SPLINE
SPL {X  -115.209, Y  +259.476, Z    +0.000, E1   +49.595, E3 +267374.990}
SPL {X  -147.344, Y  +302.806, Z    +0.000, E1   +40.158, E3 +267464.452}
SPL {X  -160.798, Y  +338.700, Z    +0.000, E1   +25.294, E3 +267463.934}
SPL {X  -163.893, Y  +354.439, Z    +0.000, E1   +16.805, E3 +267458.408}
SPL {X  -165.158, Y  +365.746, Z    +0.000, E1   +10.198, E3 +267456.351}
SPL {X  -165.639, Y  +376.620, Z    +0.000, E1    +3.186, E3 +267456.151}
SPL {X  -165.650, Y  +380.533, Z    +0.000, E1    +0.120, E3 +267455.179}
SPL {X  -165.650, Y  +383.454, Z    +0.000, E1    -2.667, E3 +267454.586}
SPL {X  -165.650, Y  +388.792, Z    +0.000, E1    -9.482, E3 +267453.680}
SPL {X  -165.650, Y  +393.970, Z    +0.000, E1   -17.146, E3 +267452.837}
SPL {X  -165.650, Y  +401.614, Z    +0.000, E1   -27.619, E3 +267453.492}
SPL {X  -165.650, Y  +418.105, Z    +0.000, E1   -49.413, E3 +267448.900}
SPL {X  -165.650, Y  +465.736, Z    +0.000, E1   -65.678, E3 +267462.642}
SPL {X  -165.650, Y  +519.483, Z    +0.000, E1   -68.357, E3 +267488.827}
SPL {X  -165.650, Y  +548.869, Z    +0.000, E1   -62.199, E3 +267544.519}
ENDSPLINE

SPLINE
SPL {X  -165.650, Y  +534.780, Z    +0.000, E1   -57.803, E3 +267558.169}
ENDSPLINE

SPLINE
SPL {X  -165.650, Y  +545.905, Z    +0.000, E1   -57.853, E3 +267572.108}
SPL {X  -165.650, Y  +553.630, Z    +0.000, E1   -57.616, E3 +267583.558}
SPL {X  -165.650, Y  +563.473, Z    +0.000, E1   -57.690, E3 +267595.922}
SPL {X  -165.650, Y  +573.011, Z    +0.000, E1   -57.610, E3 +267608.713}
SPL {X  -165.650, Y  +581.530, Z    +0.000, E1   -57.678, E3 +267619.311}
SPL {X  -165.650, Y  +589.475, Z    +0.000, E1   -57.572, E3 +267630.298}
SPL {X  -165.650, Y  +599.695, Z    +0.000, E1   -57.964, E3 +267640.914}
SPL {X  -165.650, Y  +606.915, Z    +0.000, E1   -57.651, E3 +267652.271}
SPL {X  -165.650, Y  +614.927, Z    +0.000, E1   -57.517, E3 +267663.541}
SPL {X  -165.650, Y  +624.337, Z    +0.000, E1   -57.671, E3 +267674.767}
SPL {X  -165.650, Y  +634.236, Z    +0.000, E1   -57.671, E3 +267687.617}
SPL {X  -165.650, Y  +644.287, Z    +0.000, E1   -57.872, E3 +267699.183}
SPL {X  -165.650, Y  +650.480, Z    +0.000, E1   -57.669, E3 +267708.488}
SPL {X  -165.650, Y  +657.986, Z    +0.000, E1   -57.646, E3 +267718.380}
SPL {X  -165.650, Y  +667.585, Z    +0.000, E1   -57.803, E3 +267729.776}
SPL {X  -165.650, Y  +673.199, Z    +0.000, E1   -57.412, E3 +267739.520}
SPL {X  -165.558, Y  +681.013, Z    +0.000, E1   -57.768, E3 +267747.359}
SPL {X  -165.167, Y  +688.139, Z    +0.000, E1   -57.463, E3 +267758.657}
SPL {X  -164.323, Y  +696.426, Z    +0.000, E1   -57.565, E3 +267768.644}
SPL {X  -163.313, Y  +703.224, Z    +0.000, E1   -57.403, E3 +267778.538}
SPL {X  -161.906, Y  +710.520, Z    +0.000, E1   -57.149, E3 +267789.489}
SPL {X  -160.577, Y  +716.182, Z    +0.000, E1   -56.676, E3 +267799.750}
SPL {X  -158.520, Y  +723.576, Z    +0.000, E1   -56.758, E3 +267808.795}
SPL {X  -156.858, Y  +728.749, Z    +0.000, E1   -56.333, E3 +267817.937}
SPL {X  -155.155, Y  +733.525, Z    +0.000, E1   -55.869, E3 +267826.714}
SPL {X  -153.442, Y  +737.914, Z    +0.000, E1   -55.562, E3 +267834.118}
SPL {X  -150.574, Y  +744.547, Z    +0.000, E1   -55.310, E3 +267844.101}
SPL {X  -147.713, Y  +750.471, Z    +0.000, E1   -54.514, E3 +267855.764}
SPL {X  -139.786, Y  +764.381, Z    +0.000, E1   -57.209, E3 +267859.952}
SPL {X  -110.324, Y  +799.066, Z    +0.000, E1   -54.396, E3 +267928.526}
SPL {X  -100.308, Y  +807.326, Z    +0.000, E1   -52.880, E3 +267973.093}
ENDSPLINE

SPLINE
SPL {X  -108.196, Y  +800.934, Z    +0.000, E1   -52.068, E3 +268065.420}
SPL {X  -144.673, Y  +756.182, Z    +0.000, E1   -41.752, E3 +268083.499}
SPL {X  -158.838, Y  +722.515, Z    +0.000, E1   -28.697, E3 +268082.983}
SPL {X  -163.562, Y  +701.720, Z    +0.000, E1   -18.114, E3 +268080.196}
SPL {X  -165.078, Y  +689.251, Z    +0.000, E1   -10.876, E3 +268081.748}
SPL {X  -165.596, Y  +679.730, Z    +0.000, E1    -4.777, E3 +268079.267}
SPL {X  -165.650, Y  +674.376, Z    +0.000, E1    -0.866, E3 +268079.183}
SPL {X  -165.650, Y  +672.384, Z    +0.000, E1    +0.908, E3 +268078.064}
SPL {X  -165.650, Y  +669.093, Z    +0.000, E1    +4.549, E3 +268077.915}
SPL {X  -165.650, Y  +663.273, Z    +0.000, E1   +12.448, E3 +268077.152}
SPL {X  -165.650, Y  +654.885, Z    +0.000, E1   +25.204, E3 +268075.704}
SPL {X  -165.650, Y  +641.882, Z    +0.000, E1   +46.566, E3 +268068.575}
SPL {X  -165.650, Y  +630.946, Z    +0.000, E1   +55.779, E3 +268069.250}
SPL {X  -165.650, Y  +595.858, Z    +0.000, E1   +64.262, E3 +268084.131}
SPL {X  -165.650, Y  +589.368, Z    +0.000, E1   +58.232, E3 +268104.872}
SPL {X  -165.650, Y  +491.251, Z    +0.000, E1   +65.373, E3 +268161.299}
ENDSPLINE

SPLINE
SPL {X  -165.650, Y  +516.236, Z    +0.000, E1   +58.457, E3 +268181.979}
ENDSPLINE

SPLINE
SPL {X  -165.650, Y  +506.715, Z    +0.000, E1   +58.090, E3 +268196.432}
SPL {X  -165.650, Y  +496.085, Z    +0.000, E1   +57.984, E3 +268210.680}
SPL {X  -165.650, Y  +485.167, Z    +0.000, E1   +58.003, E3 +268224.512}
ENDSPLINE

SPLINE
SPL {X  -165.650, Y  +509.193, Z    +0.000, E1   +50.604, E3 +268235.478}
ENDSPLINE

SPLINE
SPL {X  -165.650, Y  +503.302, Z    +0.000, E1   +50.402, E3 +268246.575}
SPL {X  -165.650, Y  +495.166, Z    +0.000, E1   +51.070, E3 +268256.152}
SPL {X  -165.650, Y  +485.807, Z    +0.000, E1   +51.973, E3 +268265.885}
SPL {X  -165.650, Y  +478.030, Z    +0.000, E1   +52.389, E3 +268275.691}
SPL {X  -165.650, Y  +467.527, Z    +0.000, E1   +53.334, E3 +268286.186}
SPL {X  -165.650, Y  +457.379, Z    +0.000, E1   +53.935, E3 +268297.729}
SPL {X  -165.650, Y  +444.120, Z    +0.000, E1   +54.815, E3 +268311.775}
SPL {X  -165.650, Y  +431.771, Z    +0.000, E1   +55.549, E3 +268324.604}
SPL {X  -165.650, Y  +420.799, Z    +0.000, E1   +56.452, E3 +268333.990}
SPL {X  -165.650, Y  +409.731, Z    +0.000, E1   +57.273, E3 +268343.479}
SPL {X  -165.650, Y  +399.687, Z    +0.000, E1   +57.433, E3 +268355.663}
SPL {X  -165.650, Y  +388.492, Z    +0.000, E1   +57.709, E3 +268368.376}
SPL {X  -165.650, Y  +379.894, Z    +0.000, E1   +57.709, E3 +268379.480}
SPL {X  -165.538, Y  +372.423, Z    +0.000, E1   +57.528, E3 +268390.353}
SPL {X  -164.865, Y  +362.388, Z    +0.000, E1   +57.628, E3 +268402.739}
SPL {X  -163.867, Y  +354.258, Z    +0.000, E1   +57.359, E3 +268414.956}
SPL {X  -162.678, Y  +347.264, Z    +0.000, E1   +57.150, E3 +268425.298}
SPL {X  -161.618, Y  +342.173, Z    +0.000, E1   +56.783, E3 +268434.183}
SPL {X  -159.878, Y  +335.155, Z    +0.000, E1   +56.685, E3 +268443.987}
SPL {X  -158.009, Y  +328.771, Z    +0.000, E1   +56.325, E3 +268454.346}
SPL {X  -156.065, Y  +322.971, Z    +0.000, E1   +56.177, E3 +268462.690}
SPL {X  -154.487, Y  +318.719, Z    +0.000, E1   +55.733, E3 +268470.699}
SPL {X  -151.902, Y  +312.426, Z    +0.000, E1   +55.494, E3 +268480.174}
SPL {X  -149.742, Y  +307.668, Z    +0.000, E1   +54.896, E3 +268489.386}
SPL {X  -146.487, Y  +301.160, Z    +0.000, E1   +54.808, E3 +268498.249}
SPL {X  -133.590, Y  +280.553, Z    +0.000, E1   +59.642, E3 +268499.206}
SPL {X  -112.638, Y  +257.040, Z    +0.000, E1   +51.417, E3 +268602.589}
ENDSPLINE

SPLINE
SPL {X  -115.209, Y  +259.476, Z    +0.000, E1   +49.595, E3 +268635.859}
SPL {X  -147.344, Y  +302.806, Z    +0.000, E1   +40.158, E3 +268725.322}
SPL {X  -160.798, Y  +338.700, Z    +0.000, E1   +25.294, E3 +268724.804}
SPL {X  -163.893, Y  +354.439, Z    +0.000, E1   +16.805, E3 +268719.278}
SPL {X  -165.158, Y  +365.746, Z    +0.000, E1   +10.198, E3 +268717.220}
SPL {X  -165.580, Y  +373.688, Z    +0.000, E1    +5.094, E3 +268716.957}
SPL {X  -165.650, Y  +379.719, Z    +0.000, E1    +0.894, E3 +268716.387}
SPL {X  -165.650, Y  +383.454, Z    +0.000, E1    -2.667, E3 +268715.455}
SPL {X  -165.650, Y  +387.779, Z    +0.000, E1    -8.159, E3 +268715.129}
SPL {X  -165.650, Y  +392.511, Z    +0.000, E1   -14.940, E3 +268713.620}
SPL {X  -165.650, Y  +401.614, Z    +0.000, E1   -27.619, E3 +268714.361}
SPL {X  -165.650, Y  +417.340, Z    +0.000, E1   -48.811, E3 +268709.663}
SPL {X  -165.650, Y  +462.495, Z    +0.000, E1   -65.156, E3 +268722.495}
SPL {X  -165.650, Y  +519.483, Z    +0.000, E1   -68.357, E3 +268749.696}
SPL {X  -165.650, Y  +548.869, Z    +0.000, E1   -62.199, E3 +268805.389}
ENDSPLINE

SPLINE
SPL {X  -165.650, Y  +534.780, Z    +0.000, E1   -57.803, E3 +268819.038}
ENDSPLINE

SPLINE
SPL {X  -165.650, Y  +545.905, Z    +0.000, E1   -57.853, E3 +268832.978}
SPL {X  -165.650, Y  +553.630, Z    +0.000, E1   -57.616, E3 +268844.427}
SPL {X  -165.650, Y  +563.473, Z    +0.000, E1   -57.690, E3 +268856.791}
SPL {X  -165.650, Y  +573.011, Z    +0.000, E1   -57.610, E3 +268869.583}
SPL {X  -165.650, Y  +581.530, Z    +0.000, E1   -57.678, E3 +268880.181}
SPL {X  -165.650, Y  +589.475, Z    +0.000, E1   -57.572, E3 +268891.168}
SPL {X  -165.650, Y  +599.695, Z    +0.000, E1   -57.964, E3 +268901.784}
SPL {X  -165.650, Y  +606.915, Z    +0.000, E1   -57.651, E3 +268913.140}
SPL {X  -165.650, Y  +614.927, Z    +0.000, E1   -57.517, E3 +268924.410}
SPL {X  -165.650, Y  +624.337, Z    +0.000, E1   -57.671, E3 +268935.636}
SPL {X  -165.650, Y  +634.236, Z    +0.000, E1   -57.671, E3 +268948.486}
SPL {X  -165.650, Y  +647.519, Z    +0.000, E1   -57.817, E3 +268964.814}
SPL {X  -165.650, Y  +657.986, Z    +0.000, E1   -57.646, E3 +268979.249}
SPL {X  -165.650, Y  +667.585, Z    +0.000, E1   -57.803, E3 +268990.645}
SPL {X  -165.634, Y  +677.794, Z    +0.000, E1   -57.650, E3 +269004.947}
SPL {X  -165.167, Y  +688.139, Z    +0.000, E1   -57.463, E3 +269019.527}
SPL {X  -164.009, Y  +698.761, Z    +0.000, E1   -57.613, E3 +269032.300}
SPL {X  -162.382, Y  +708.242, Z    +0.000, E1   -57.205, E3 +269047.226}
SPL {X  -160.577, Y  +716.182, Z    +0.000, E1   -56.676, E3 +269060.619}
SPL {X  -158.520, Y  +723.576, Z    +0.000, E1   -56.758, E3 +269069.664}
SPL {X  -156.858, Y  +728.749, Z    +0.000, E1   -56.333, E3 +269078.807}
SPL {X  -155.155, Y  +733.525, Z    +0.000, E1   -55.869, E3 +269087.583}
SPL {X  -153.442, Y  +737.914, Z    +0.000, E1   -55.562, E3 +269094.988}
SPL {X  -150.574, Y  +744.547, Z    +0.000, E1   -55.310, E3 +269104.971}
SPL {X  -147.713, Y  +750.471, Z    +0.000, E1   -54.514, E3 +269116.633}
SPL {X  -139.786, Y  +764.381, Z    +0.000, E1   -57.209, E3 +269120.821}
SPL {X  -110.324, Y  +799.066, Z    +0.000, E1   -54.396, E3 +269189.396}
SPL {X  -100.308, Y  +807.326, Z    +0.000, E1   -52.880, E3 +269233.963}
ENDSPLINE

SPLINE
SPL {X  -108.196, Y  +800.934, Z    +0.000, E1   -52.068, E3 +269326.289}
SPL {X  -144.673, Y  +756.182, Z    +0.000, E1   -41.752, E3 +269344.368}
SPL {X  -158.838, Y  +722.515, Z    +0.000, E1   -28.697, E3 +269343.852}
SPL {X  -163.562, Y  +701.720, Z    +0.000, E1   -18.114, E3 +269341.066}
SPL {X  -165.380, Y  +684.954, Z    +0.000, E1    -8.247, E3 +269341.248}
SPL {X  -165.650, Y  +675.104, Z    +0.000, E1    -1.512, E3 +269340.043}
SPL {X  -165.650, Y  +672.384, Z    +0.000, E1    +0.908, E3 +269338.933}
SPL {X  -165.650, Y  +669.968, Z    +0.000, E1    +3.584, E3 +269338.749}
SPL {X  -165.650, Y  +666.667, Z    +0.000, E1    +7.761, E3 +269338.428}
SPL {X  -165.650, Y  +662.028, Z    +0.000, E1   +14.359, E3 +269338.058}
SPL {X  -165.650, Y  +654.885, Z    +0.000, E1   +25.204, E3 +269336.574}
SPL {X  -165.650, Y  +641.882, Z    +0.000, E1   +46.566, E3 +269329.445}
SPL {X  -165.650, Y  +630.946, Z    +0.000, E1   +55.779, E3 +269330.119}
SPL {X  -165.650, Y  +590.135, Z    +0.000, E1   +59.110, E3 +269362.739}
SPL {X  -165.650, Y  +491.251, Z    +0.000, E1   +65.373, E3 +269422.168}
ENDSPLINE

SPLINE
SPL {X  -165.650, Y  +516.236, Z    +0.000, E1   +58.457, E3 +269442.849}
ENDSPLINE

SPLINE
SPL {X  -165.650, Y  +506.715, Z    +0.000, E1   +58.090, E3 +269457.302}
SPL {X  -165.650, Y  +496.085, Z    +0.000, E1   +57.984, E3 +269471.549}
SPL {X  -165.650, Y  +485.167, Z    +0.000, E1   +58.003, E3 +269485.381}
ENDSPLINE

SPLINE
SPL {X  -165.650, Y  +505.180, Z    +0.000, E1   +52.333, E3 +269492.133}
SPL {X  -165.650, Y  +506.534, Z    +0.000, E1   +50.148, E3 +269503.593}
ENDSPLINE

SPLINE
SPL {X  -165.650, Y  +495.166, Z    +0.000, E1   +51.070, E3 +269517.021}
SPL {X  -165.650, Y  +485.807, Z    +0.000, E1   +51.973, E3 +269526.754}
SPL {X  -165.650, Y  +475.672, Z    +0.000, E1   +52.573, E3 +269539.208}
SPL {X  -165.650, Y  +459.814, Z    +0.000, E1   +53.888, E3 +269555.397}
SPL {X  -165.650, Y  +448.876, Z    +0.000, E1   +54.452, E3 +269567.892}
SPL {X  -165.650, Y  +440.843, Z    +0.000, E1   +55.023, E3 +269575.956}
SPL {X  -165.650, Y  +431.771, Z    +0.000, E1   +55.549, E3 +269585.474}
SPL {X  -165.650, Y  +420.799, Z    +0.000, E1   +56.452, E3 +269594.860}
SPL {X  -165.650, Y  +409.731, Z    +0.000, E1   +57.273, E3 +269604.348}
SPL {X  -165.650, Y  +399.687, Z    +0.000, E1   +57.433, E3 +269616.533}
SPL {X  -165.650, Y  +388.492, Z    +0.000, E1   +57.709, E3 +269629.246}
SPL {X  -165.650, Y  +379.894, Z    +0.000, E1   +57.709, E3 +269640.350}
SPL {X  -165.538, Y  +372.423, Z    +0.000, E1   +57.528, E3 +269651.222}
SPL {X  -164.865, Y  +362.388, Z    +0.000, E1   +57.628, E3 +269663.609}
SPL {X  -163.867, Y  +354.258, Z    +0.000, E1   +57.359, E3 +269675.826}
SPL {X  -162.678, Y  +347.264, Z    +0.000, E1   +57.150, E3 +269686.167}
SPL {X  -161.618, Y  +342.173, Z    +0.000, E1   +56.783, E3 +269695.053}
SPL {X  -159.878, Y  +335.155, Z    +0.000, E1   +56.685, E3 +269704.856}
SPL {X  -158.009, Y  +328.771, Z    +0.000, E1   +56.325, E3 +269715.216}
SPL {X  -156.065, Y  +322.971, Z    +0.000, E1   +56.177, E3 +269723.560}
SPL {X  -153.731, Y  +316.803, Z    +0.000, E1   +55.737, E3 +269734.136}
SPL {X  -150.320, Y  +308.902, Z    +0.000, E1   +55.085, E3 +269747.832}
SPL {X  -146.487, Y  +301.160, Z    +0.000, E1   +54.808, E3 +269759.118}
SPL {X  -133.590, Y  +280.553, Z    +0.000, E1   +59.642, E3 +269760.075}
SPL {X  -112.638, Y  +257.040, Z    +0.000, E1   +51.417, E3 +269863.459}
ENDSPLINE

SPLINE
SPL {X  -115.209, Y  +259.476, Z    +0.000, E1   +49.595, E3 +269896.729}
SPL {X  -147.344, Y  +302.806, Z    +0.000, E1   +40.158, E3 +269986.191}
SPL {X  -160.798, Y  +338.700, Z    +0.000, E1   +25.294, E3 +269985.673}
SPL {X  -163.893, Y  +354.439, Z    +0.000, E1   +16.805, E3 +269980.147}
SPL {X  -165.158, Y  +365.746, Z    +0.000, E1   +10.198, E3 +269978.090}
SPL {X  -165.639, Y  +376.620, Z    +0.000, E1    +3.186, E3 +269977.890}
SPL {X  -165.650, Y  +380.533, Z    +0.000, E1    +0.120, E3 +269976.918}
SPL {X  -165.650, Y  +382.353, Z    +0.000, E1    -1.616, E3 +269976.499}
SPL {X  -165.650, Y  +386.363, Z    +0.000, E1    -6.162, E3 +269976.049}
SPL {X  -165.650, Y  +392.511, Z    +0.000, E1   -14.940, E3 +269974.489}
SPL {X  -165.650, Y  +401.614, Z    +0.000, E1   -27.619, E3 +269975.231}
SPL {X  -165.650, Y  +418.105, Z    +0.000, E1   -49.413, E3 +269970.639}
SPL {X  -165.650, Y  +465.736, Z    +0.000, E1   -65.678, E3 +269984.381}
SPL {X  -165.650, Y  +519.483, Z    +0.000, E1   -68.357, E3 +270010.566}
SPL {X  -165.650, Y  +548.869, Z    +0.000, E1   -62.199, E3 +270066.259}
ENDSPLINE

SPLINE
SPL {X  -165.650, Y  +534.780, Z    +0.000, E1   -57.803, E3 +270079.908}
ENDSPLINE

SPLINE
SPL {X  -165.650, Y  +545.905, Z    +0.000, E1   -57.853, E3 +270093.847}
SPL {X  -165.650, Y  +555.746, Z    +0.000, E1   -57.571, E3 +270108.485}
SPL {X  -165.650, Y  +566.557, Z    +0.000, E1   -57.834, E3 +270120.613}
SPL {X  -165.650, Y  +573.011, Z    +0.000, E1   -57.610, E3 +270130.452}
SPL {X  -165.650, Y  +581.530, Z    +0.000, E1   -57.678, E3 +270141.050}
SPL {X  -165.650, Y  +589.475, Z    +0.000, E1   -57.572, E3 +270152.037}
SPL {X  -165.650, Y  +599.695, Z    +0.000, E1   -57.964, E3 +270162.653}
SPL {X  -165.650, Y  +606.915, Z    +0.000, E1   -57.651, E3 +270174.010}
SPL {X  -165.650, Y  +614.927, Z    +0.000, E1   -57.517, E3 +270185.280}
SPL {X  -165.650, Y  +624.337, Z    +0.000, E1   -57.671, E3 +270196.506}
SPL {X  -165.650, Y  +634.236, Z    +0.000, E1   -57.671, E3 +270209.356}
SPL {X  -165.650, Y  +644.287, Z    +0.000, E1   -57.872, E3 +270220.922}
SPL {X  -165.650, Y  +650.480, Z    +0.000, E1   -57.669, E3 +270230.227}
SPL {X  -165.650, Y  +657.986, Z    +0.000, E1   -57.646, E3 +270240.119}
SPL {X  -165.650, Y  +667.585, Z    +0.000, E1   -57.803, E3 +270251.515}
SPL {X  -165.650, Y  +673.199, Z    +0.000, E1   -57.412, E3 +270261.259}
SPL {X  -165.558, Y  +681.013, Z    +0.000, E1   -57.768, E3 +270269.098}
SPL {X  -165.167, Y  +688.139, Z    +0.000, E1   -57.463, E3 +270280.396}
SPL {X  -164.009, Y  +698.761, Z    +0.000, E1   -57.613, E3 +270293.169}
SPL {X  -162.382, Y  +708.242, Z    +0.000, E1   -57.205, E3 +270308.095}
SPL {X  -160.577, Y  +716.182, Z    +0.000, E1   -56.676, E3 +270321.489}
SPL {X  -158.520, Y  +723.576, Z    +0.000, E1   -56.758, E3 +270330.534}
SPL {X  -156.858, Y  +728.749, Z    +0.000, E1   -56.333, E3 +270339.676}
SPL {X  -155.155, Y  +733.525, Z    +0.000, E1   -55.869, E3 +270348.453}
SPL {X  -152.530, Y  +740.111, Z    +0.000, E1   -55.545, E3 +270358.929}
SPL {X  -149.838, Y  +746.130, Z    +0.000, E1   -55.135, E3 +270368.649}
SPL {X  -147.713, Y  +750.471, Z    +0.000, E1   -54.514, E3 +270377.503}
SPL {X  -139.786, Y  +764.381, Z    +0.000, E1   -57.209, E3 +270381.691}
SPL {X  -110.324, Y  +799.066, Z    +0.000, E1   -54.396, E3 +270450.265}
SPL {X  -100.308, Y  +807.326, Z    +0.000, E1   -52.880, E3 +270494.832}
ENDSPLINE

SPLINE
SPL {X  -108.196, Y  +800.934, Z    +0.000, E1   -52.068, E3 +270587.159}
SPL {X  -147.753, Y  +750.393, Z    +0.000, E1   -39.863, E3 +270605.381}
SPL {X  -161.414, Y  +712.720, Z    +0.000, E1   -24.024, E3 +270604.723}
SPL {X  -164.278, Y  +696.774, Z    +0.000, E1   -15.225, E3 +270599.335}
SPL {X  -165.380, Y  +684.954, Z    +0.000, E1    -8.247, E3 +270602.118}
SPL {X  -165.650, Y  +675.104, Z    +0.000, E1    -1.512, E3 +270600.913}
SPL {X  -165.650, Y  +672.384, Z    +0.000, E1    +0.908, E3 +270599.803}
SPL {X  -165.650, Y  +669.093, Z    +0.000, E1    +4.549, E3 +270599.654}
SPL {X  -165.650, Y  +663.273, Z    +0.000, E1   +12.448, E3 +270598.891}
SPL {X  -165.650, Y  +657.199, Z    +0.000, E1   +21.720, E3 +270598.161}
SPL {X  -165.650, Y  +652.963, Z    +0.000, E1   +28.395, E3 +270596.846}
SPL {X  -165.650, Y  +641.882, Z    +0.000, E1   +46.566, E3 +270590.314}
SPL {X  -165.650, Y  +630.946, Z    +0.000, E1   +55.779, E3 +270590.989}
SPL {X  -165.650, Y  +590.135, Z    +0.000, E1   +59.110, E3 +270623.609}
SPL {X  -165.650, Y  +491.251, Z    +0.000, E1   +65.373, E3 +270683.038}
ENDSPLINE

SPLINE
SPL {X  -165.650, Y  +516.236, Z    +0.000, E1   +58.457, E3 +270703.718}
ENDSPLINE

SPLINE
SPL {X  -165.650, Y  +506.715, Z    +0.000, E1   +58.090, E3 +270718.171}
SPL {X  -165.650, Y  +496.085, Z    +0.000, E1   +57.984, E3 +270732.419}
SPL {X  -165.650, Y  +485.167, Z    +0.000, E1   +58.003, E3 +270746.251}
ENDSPLINE

SPLINE
SPL {X  -165.650, Y  +509.193, Z    +0.000, E1   +50.604, E3 +270757.218}
ENDSPLINE

SPLINE
SPL {X  -165.650, Y  +503.302, Z    +0.000, E1   +50.402, E3 +270768.314}
SPL {X  -165.650, Y  +495.166, Z    +0.000, E1   +51.070, E3 +270777.891}
SPL {X  -165.650, Y  +485.807, Z    +0.000, E1   +51.973, E3 +270787.624}
SPL {X  -165.650, Y  +478.030, Z    +0.000, E1   +52.389, E3 +270797.431}
SPL {X  -165.650, Y  +467.527, Z    +0.000, E1   +53.334, E3 +270807.925}
SPL {X  -165.650, Y  +457.379, Z    +0.000, E1   +53.935, E3 +270819.468}
SPL {X  -165.650, Y  +444.120, Z    +0.000, E1   +54.815, E3 +270833.514}
SPL {X  -165.650, Y  +431.771, Z    +0.000, E1   +55.549, E3 +270846.344}
SPL {X  -165.650, Y  +420.799, Z    +0.000, E1   +56.452, E3 +270855.729}
SPL {X  -165.650, Y  +409.731, Z    +0.000, E1   +57.273, E3 +270865.218}
SPL {X  -165.650, Y  +399.687, Z    +0.000, E1   +57.433, E3 +270877.402}
SPL {X  -165.650, Y  +388.492, Z    +0.000, E1   +57.709, E3 +270890.115}
SPL {X  -165.650, Y  +379.894, Z    +0.000, E1   +57.709, E3 +270901.219}
SPL {X  -165.538, Y  +372.423, Z    +0.000, E1   +57.528, E3 +270912.092}
SPL {X  -164.865, Y  +362.388, Z    +0.000, E1   +57.628, E3 +270924.478}
SPL {X  -163.867, Y  +354.258, Z    +0.000, E1   +57.359, E3 +270936.695}
SPL {X  -162.678, Y  +347.264, Z    +0.000, E1   +57.150, E3 +270947.037}
SPL {X  -161.618, Y  +342.173, Z    +0.000, E1   +56.783, E3 +270955.922}
SPL {X  -159.878, Y  +335.155, Z    +0.000, E1   +56.685, E3 +270965.726}
SPL {X  -158.009, Y  +328.771, Z    +0.000, E1   +56.325, E3 +270976.086}
SPL {X  -156.065, Y  +322.971, Z    +0.000, E1   +56.177, E3 +270984.429}
SPL {X  -154.487, Y  +318.719, Z    +0.000, E1   +55.733, E3 +270992.438}
SPL {X  -151.902, Y  +312.426, Z    +0.000, E1   +55.494, E3 +271001.913}
SPL {X  -149.742, Y  +307.668, Z    +0.000, E1   +54.896, E3 +271011.125}
SPL {X  -146.487, Y  +301.160, Z    +0.000, E1   +54.808, E3 +271019.988}
SPL {X  -133.590, Y  +280.553, Z    +0.000, E1   +59.642, E3 +271020.945}
SPL {X  -112.638, Y  +257.040, Z    +0.000, E1   +51.417, E3 +271124.328}
ENDSPLINE

SPLINE
SPL {X  -115.209, Y  +259.476, Z    +0.000, E1   +49.595, E3 +271157.599}
SPL {X  -147.344, Y  +302.806, Z    +0.000, E1   +40.158, E3 +271247.061}
SPL {X  -160.798, Y  +338.700, Z    +0.000, E1   +25.294, E3 +271246.543}
SPL {X  -163.893, Y  +354.439, Z    +0.000, E1   +16.805, E3 +271241.017}
SPL {X  -165.158, Y  +365.746, Z    +0.000, E1   +10.198, E3 +271238.959}
SPL {X  -165.580, Y  +373.688, Z    +0.000, E1    +5.094, E3 +271238.696}
SPL {X  -165.650, Y  +378.140, Z    +0.000, E1    +1.996, E3 +271238.783}
SPL {X  -165.650, Y  +381.477, Z    +0.000, E1    -0.622, E3 +271237.570}
SPL {X  -165.650, Y  +384.861, Z    +0.000, E1    -4.465, E3 +271236.973}
SPL {X  -165.650, Y  +388.792, Z    +0.000, E1    -9.482, E3 +271236.289}
SPL {X  -165.650, Y  +396.421, Z    +0.000, E1   -20.352, E3 +271236.086}
SPL {X  -165.650, Y  +404.249, Z    +0.000, E1   -31.650, E3 +271235.465}
SPL {X  -165.650, Y  +417.340, Z    +0.000, E1   -48.811, E3 +271231.402}
SPL {X  -165.650, Y  +462.495, Z    +0.000, E1   -65.156, E3 +271244.234}
SPL {X  -165.650, Y  +519.483, Z    +0.000, E1   -68.357, E3 +271271.436}
SPL {X  -165.650, Y  +548.869, Z    +0.000, E1   -62.199, E3 +271327.128}
ENDSPLINE

SPLINE
SPL {X  -165.650, Y  +530.735, Z    +0.000, E1   -57.778, E3 +271335.552}
ENDSPLINE

SPLINE
SPL {X  -165.650, Y  +536.777, Z    +0.000, E1   -57.774, E3 +271343.429}
SPL {X  -165.650, Y  +545.905, Z    +0.000, E1   -57.853, E3 +271354.717}
SPL {X  -165.650, Y  +553.630, Z    +0.000, E1   -57.616, E3 +271366.166}
SPL {X  -165.650, Y  +563.473, Z    +0.000, E1   -57.690, E3 +271378.531}
SPL {X  -165.650, Y  +573.011, Z    +0.000, E1   -57.610, E3 +271391.322}
SPL {X  -165.650, Y  +581.530, Z    +0.000, E1   -57.678, E3 +271401.920}
SPL {X  -165.650, Y  +589.475, Z    +0.000, E1   -57.572, E3 +271412.907}
SPL {X  -165.650, Y  +599.695, Z    +0.000, E1   -57.964, E3 +271423.523}
SPL {X  -165.650, Y  +606.915, Z    +0.000, E1   -57.651, E3 +271434.880}
SPL {X  -165.650, Y  +614.927, Z    +0.000, E1   -57.517, E3 +271446.149}
SPL {X  -165.650, Y  +624.337, Z    +0.000, E1   -57.671, E3 +271457.375}
SPL {X  -165.650, Y  +634.236, Z    +0.000, E1   -57.671, E3 +271470.226}
SPL {X  -165.650, Y  +647.519, Z    +0.000, E1   -57.817, E3 +271486.553}
SPL {X  -165.650, Y  +657.986, Z    +0.000, E1   -57.646, E3 +271500.988}
SPL {X  -165.650, Y  +667.585, Z    +0.000, E1   -57.803, E3 +271512.384}
SPL {X  -165.634, Y  +677.794, Z    +0.000, E1   -57.650, E3 +271526.686}
SPL {X  -165.167, Y  +688.139, Z    +0.000, E1   -57.463, E3 +271541.266}
SPL {X  -164.009, Y  +698.761, Z    +0.000, E1   -57.613, E3 +271554.039}
SPL {X  -162.382, Y  +708.242, Z    +0.000, E1   -57.205, E3 +271568.965}
SPL {X  -160.577, Y  +716.182, Z    +0.000, E1   -56.676, E3 +271582.359}
SPL {X  -158.520, Y  +723.576, Z    +0.000, E1   -56.758, E3 +271591.403}
SPL {X  -156.858, Y  +728.749, Z    +0.000, E1   -56.333, E3 +271600.546}
SPL {X  -155.155, Y  +733.525, Z    +0.000, E1   -55.869, E3 +271609.323}
SPL {X  -153.442, Y  +737.914, Z    +0.000, E1   -55.562, E3 +271616.727}
SPL {X  -150.574, Y  +744.547, Z    +0.000, E1   -55.310, E3 +271626.710}
SPL {X  -148.396, Y  +749.110, Z    +0.000, E1   -54.616, E3 +271636.003}
SPL {X  -146.339, Y  +753.120, Z    +0.000, E1   -54.477, E3 +271641.889}
SPL {X  -137.656, Y  +767.645, Z    +0.000, E1   -58.229, E3 +271641.599}
SPL {X  -110.324, Y  +799.066, Z    +0.000, E1   -54.396, E3 +271711.135}
SPL {X  -100.308, Y  +807.326, Z    +0.000, E1   -52.880, E3 +271755.702}
ENDSPLINE

SPLINE
SPL {X  -108.196, Y  +800.934, Z    +0.000, E1   -52.068, E3 +271848.028}
SPL {X  -147.753, Y  +750.393, Z    +0.000, E1   -39.863, E3 +271866.251}
SPL {X  -161.414, Y  +712.720, Z    +0.000, E1   -24.024, E3 +271865.593}
SPL {X  -164.278, Y  +696.774, Z    +0.000, E1   -15.225, E3 +271860.205}
SPL {X  -165.380, Y  +684.954, Z    +0.000, E1    -8.247, E3 +271862.988}
SPL {X  -165.650, Y  +675.104, Z    +0.000, E1    -1.512, E3 +271861.782}
SPL {X  -165.650, Y  +672.384, Z    +0.000, E1    +0.908, E3 +271860.672}
SPL {X  -165.650, Y  +669.968, Z    +0.000, E1    +3.584, E3 +271860.488}
SPL {X  -165.650, Y  +666.667, Z    +0.000, E1    +7.761, E3 +271860.167}
SPL {X  -165.650, Y  +662.028, Z    +0.000, E1   +14.359, E3 +271859.797}
SPL {X  -165.650, Y  +654.885, Z    +0.000, E1   +25.204, E3 +271858.313}
SPL {X  -165.650, Y  +641.882, Z    +0.000, E1   +46.566, E3 +271851.184}
SPL {X  -165.650, Y  +630.946, Z    +0.000, E1   +55.779, E3 +271851.859}
SPL {X  -165.650, Y  +590.135, Z    +0.000, E1   +59.110, E3 +271884.478}
SPL {X  -165.650, Y  +491.251, Z    +0.000, E1   +65.373, E3 +271943.907}
ENDSPLINE

SPLINE
SPL {X  -165.650, Y  +516.236, Z    +0.000, E1   +58.457, E3 +271964.588}
ENDSPLINE

SPLINE
SPL {X  -165.650, Y  +506.715, Z    +0.000, E1   +58.090, E3 +271979.041}
SPL {X  -165.650, Y  +499.697, Z    +0.000, E1   +57.857, E3 +271989.384}
SPL {X  -165.650, Y  +493.307, Z    +0.000, E1   +58.045, E3 +271996.342}
SPL {X  -165.650, Y  +485.167, Z    +0.000, E1   +58.003, E3 +272007.120}
ENDSPLINE

SPLINE
SPL {X  -165.650, Y  +505.180, Z    +0.000, E1   +52.333, E3 +272013.872}
SPL {X  -165.650, Y  +506.534, Z    +0.000, E1   +50.148, E3 +272025.332}
ENDSPLINE

SPLINE
SPL {X  -165.650, Y  +495.166, Z    +0.000, E1   +51.070, E3 +272038.760}
SPL {X  -165.650, Y  +485.807, Z    +0.000, E1   +51.973, E3 +272048.493}
SPL {X  -165.650, Y  +478.030, Z    +0.000, E1   +52.389, E3 +272058.300}
SPL {X  -165.650, Y  +467.527, Z    +0.000, E1   +53.334, E3 +272068.794}
SPL {X  -165.650, Y  +457.379, Z    +0.000, E1   +53.935, E3 +272080.338}
SPL {X  -165.650, Y  +444.120, Z    +0.000, E1   +54.815, E3 +272094.383}
SPL {X  -165.650, Y  +431.771, Z    +0.000, E1   +55.549, E3 +272107.213}
SPL {X  -165.650, Y  +420.799, Z    +0.000, E1   +56.452, E3 +272116.599}
SPL {X  -165.650, Y  +409.731, Z    +0.000, E1   +57.273, E3 +272126.087}
SPL {X  -165.650, Y  +399.687, Z    +0.000, E1   +57.433, E3 +272138.272}
SPL {X  -165.650, Y  +388.492, Z    +0.000, E1   +57.709, E3 +272150.985}
SPL {X  -165.650, Y  +379.894, Z    +0.000, E1   +57.709, E3 +272162.089}
SPL {X  -165.538, Y  +372.423, Z    +0.000, E1   +57.528, E3 +272172.961}
SPL {X  -164.865, Y  +362.388, Z    +0.000, E1   +57.628, E3 +272185.348}
SPL {X  -163.867, Y  +354.258, Z    +0.000, E1   +57.359, E3 +272197.565}
SPL {X  -162.678, Y  +347.264, Z    +0.000, E1   +57.150, E3 +272207.906}
SPL {X  -161.618, Y  +342.173, Z    +0.000, E1   +56.783, E3 +272216.792}
SPL {X  -159.878, Y  +335.155, Z    +0.000, E1   +56.685, E3 +272226.595}
SPL {X  -158.009, Y  +328.771, Z    +0.000, E1   +56.325, E3 +272236.955}
SPL {X  -156.065, Y  +322.971, Z    +0.000, E1   +56.177, E3 +272245.299}
SPL {X  -154.487, Y  +318.719, Z    +0.000, E1   +55.733, E3 +272253.308}
SPL {X  -151.902, Y  +312.426, Z    +0.000, E1   +55.494, E3 +272262.783}
SPL {X  -148.935, Y  +305.985, Z    +0.000, E1   +54.737, E3 +272275.159}
SPL {X  -144.791, Y  +298.030, Z    +0.000, E1   +55.214, E3 +272282.892}
SPL {X  -133.590, Y  +280.553, Z    +0.000, E1   +59.642, E3 +272281.814}
SPL {X  -112.638, Y  +257.040, Z    +0.000, E1   +51.417, E3 +272385.198}
ENDSPLINE

SPLINE
SPL {X  -115.209, Y  +259.476, Z    +0.000, E1   +49.595, E3 +272418.468}
SPL {X  -147.344, Y  +302.806, Z    +0.000, E1   +40.158, E3 +272507.930}
SPL {X  -160.798, Y  +338.700, Z    +0.000, E1   +25.294, E3 +272507.412}
SPL {X  -163.893, Y  +354.439, Z    +0.000, E1   +16.805, E3 +272501.886}
SPL {X  -165.158, Y  +365.746, Z    +0.000, E1   +10.198, E3 +272499.829}
SPL {X  -165.639, Y  +376.620, Z    +0.000, E1    +3.186, E3 +272499.629}
SPL {X  -165.650, Y  +380.533, Z    +0.000, E1    +0.120, E3 +272498.657}
SPL {X  -165.650, Y  +383.454, Z    +0.000, E1    -2.667, E3 +272498.064}
SPL {X  -165.650, Y  +388.792, Z    +0.000, E1    -9.482, E3 +272497.158}
SPL {X  -165.650, Y  +396.421, Z    +0.000, E1   -20.352, E3 +272496.956}
SPL {X  -165.650, Y  +404.249, Z    +0.000, E1   -31.650, E3 +272496.335}
SPL {X  -165.650, Y  +418.105, Z    +0.000, E1   -49.413, E3 +272492.378}
SPL {X  -165.650, Y  +465.736, Z    +0.000, E1   -65.678, E3 +272506.120}
SPL {X  -165.650, Y  +519.483, Z    +0.000, E1   -68.357, E3 +272532.305}
SPL {X  -165.650, Y  +548.869, Z    +0.000, E1   -62.199, E3 +272587.998}
ENDSPLINE

SPLINE
SPL {X  -165.650, Y  +530.735, Z    +0.000, E1   -57.778, E3 +272596.421}
ENDSPLINE

SPLINE
SPL {X  -165.650, Y  +536.777, Z    +0.000, E1   -57.774, E3 +272604.298}
SPL {X  -165.650, Y  +545.905, Z    +0.000, E1   -57.853, E3 +272615.586}
SPL {X  -165.650, Y  +553.630, Z    +0.000, E1   -57.616, E3 +272627.036}
SPL {X  -165.650, Y  +563.473, Z    +0.000, E1   -57.690, E3 +272639.400}
SPL {X  -165.650, Y  +573.011, Z    +0.000, E1   -57.610, E3 +272652.191}
SPL {X  -165.650, Y  +581.530, Z    +0.000, E1   -57.678, E3 +272662.789}
SPL {X  -165.650, Y  +589.475, Z    +0.000, E1   -57.572, E3 +272673.776}
SPL {X  -165.650, Y  +599.695, Z    +0.000, E1   -57.964, E3 +272684.392}
SPL {X  -165.650, Y  +606.915, Z    +0.000, E1   -57.651, E3 +272695.749}
SPL {X  -165.650, Y  +614.927, Z    +0.000, E1   -57.517, E3 +272707.019}
SPL {X  -165.650, Y  +624.337, Z    +0.000, E1   -57.671, E3 +272718.245}
SPL {X  -165.650, Y  +634.236, Z    +0.000, E1   -57.671, E3 +272731.095}
SPL {X  -165.650, Y  +647.519, Z    +0.000, E1   -57.817, E3 +272747.422}
SPL {X  -165.650, Y  +657.986, Z    +0.000, E1   -57.646, E3 +272761.858}
SPL {X  -165.650, Y  +667.585, Z    +0.000, E1   -57.803, E3 +272773.254}
SPL {X  -165.634, Y  +677.794, Z    +0.000, E1   -57.650, E3 +272787.556}
SPL {X  -165.167, Y  +688.139, Z    +0.000, E1   -57.463, E3 +272802.135}
SPL {X  -164.323, Y  +696.426, Z    +0.000, E1   -57.565, E3 +272812.122}
SPL {X  -163.313, Y  +703.224, Z    +0.000, E1   -57.403, E3 +272822.016}
SPL {X  -161.906, Y  +710.520, Z    +0.000, E1   -57.149, E3 +272832.967}
SPL {X  -160.577, Y  +716.182, Z    +0.000, E1   -56.676, E3 +272843.228}
SPL {X  -158.520, Y  +723.576, Z    +0.000, E1   -56.758, E3 +272852.273}
SPL {X  -156.858, Y  +728.749, Z    +0.000, E1   -56.333, E3 +272861.416}
SPL {X  -155.155, Y  +733.525, Z    +0.000, E1   -55.869, E3 +272870.192}
SPL {X  -153.442, Y  +737.914, Z    +0.000, E1   -55.562, E3 +272877.597}
SPL {X  -150.574, Y  +744.547, Z    +0.000, E1   -55.310, E3 +272887.579}
SPL {X  -147.713, Y  +750.471, Z    +0.000, E1   -54.514, E3 +272899.242}
SPL {X  -139.786, Y  +764.381, Z    +0.000, E1   -57.209, E3 +272903.430}
SPL {X  -110.324, Y  +799.066, Z    +0.000, E1   -54.396, E3 +272972.004}
SPL {X  -100.308, Y  +807.326, Z    +0.000, E1   -52.880, E3 +273016.571}
ENDSPLINE

SPLINE
SPL {X  -108.196, Y  +800.934, Z    +0.000, E1   -52.068, E3 +273108.898}
SPL {X  -144.673, Y  +756.182, Z    +0.000, E1   -41.752, E3 +273126.977}
SPL {X  -158.838, Y  +722.515, Z    +0.000, E1   -28.697, E3 +273126.461}
SPL {X  -163.562, Y  +701.720, Z    +0.000, E1   -18.114, E3 +273123.675}
SPL {X  -165.078, Y  +689.251, Z    +0.000, E1   -10.876, E3 +273125.226}
SPL {X  -165.596, Y  +679.730, Z    +0.000, E1    -4.777, E3 +273122.745}
SPL {X  -165.650, Y  +674.376, Z    +0.000, E1    -0.866, E3 +273122.661}
SPL {X  -165.650, Y  +672.384, Z    +0.000, E1    +0.908, E3 +273121.542}
SPL {X  -165.650, Y  +669.093, Z    +0.000, E1    +4.549, E3 +273121.393}
SPL {X  -165.650, Y  +663.273, Z    +0.000, E1   +12.448, E3 +273120.631}
SPL {X  -165.650, Y  +654.885, Z    +0.000, E1   +25.204, E3 +273119.182}
SPL {X  -165.650, Y  +641.882, Z    +0.000, E1   +46.566, E3 +273112.053}
SPL {X  -165.650, Y  +630.946, Z    +0.000, E1   +55.779, E3 +273112.728}
SPL {X  -165.650, Y  +595.858, Z    +0.000, E1   +64.262, E3 +273127.609}
SPL {X  -165.650, Y  +589.368, Z    +0.000, E1   +58.232, E3 +273148.350}
SPL {X  -165.650, Y  +491.251, Z    +0.000, E1   +65.373, E3 +273204.777}
ENDSPLINE

SPLINE
SPL {X  -165.650, Y  +516.236, Z    +0.000, E1   +58.457, E3 +273225.458}
ENDSPLINE

SPLINE
SPL {X  -165.650, Y  +506.715, Z    +0.000, E1   +58.090, E3 +273239.911}
SPL {X  -165.650, Y  +496.085, Z    +0.000, E1   +57.984, E3 +273254.158}
SPL {X  -165.650, Y  +485.167, Z    +0.000, E1   +58.003, E3 +273267.990}
ENDSPLINE

SPLINE
SPL {X  -165.650, Y  +509.193, Z    +0.000, E1   +50.604, E3 +273278.957}
ENDSPLINE

SPLINE
SPL {X  -165.650, Y  +503.302, Z    +0.000, E1   +50.402, E3 +273290.053}
SPL {X  -165.650, Y  +495.166, Z    +0.000, E1   +51.070, E3 +273299.630}
SPL {X  -165.650, Y  +485.807, Z    +0.000, E1   +51.973, E3 +273309.363}
SPL {X  -165.650, Y  +478.030, Z    +0.000, E1   +52.389, E3 +273319.170}
SPL {X  -165.650, Y  +467.527, Z    +0.000, E1   +53.334, E3 +273329.664}
SPL {X  -165.650, Y  +457.379, Z    +0.000, E1   +53.935, E3 +273341.207}
SPL {X  -165.650, Y  +444.120, Z    +0.000, E1   +54.815, E3 +273355.253}
SPL {X  -165.650, Y  +431.771, Z    +0.000, E1   +55.549, E3 +273368.083}
SPL {X  -165.650, Y  +420.799, Z    +0.000, E1   +56.452, E3 +273377.469}
SPL {X  -165.650, Y  +406.746, Z    +0.000, E1   +57.489, E3 +273389.513}
ENDSPLINE

SPLINE
SPL {X  -165.650, Y  +413.842, Z    +0.000, E1   +53.687, E3 +273403.647}
ENDSPLINE

SPLINE
SPL {X  -165.650, Y  +405.379, Z    +0.000, E1   +53.922, E3 +273414.760}
SPL {X  -165.650, Y  +400.791, Z    +0.000, E1   +53.827, E3 +273422.173}
SPL {X  -165.650, Y  +391.401, Z    +0.000, E1   +53.934, E3 +273435.773}
SPL {X  -165.650, Y  +378.987, Z    +0.000, E1   +53.974, E3 +273453.969}
SPL {X  -165.408, Y  +369.556, Z    +0.000, E1   +53.942, E3 +273468.061}
SPL {X  -164.927, Y  +363.041, Z    +0.000, E1   +53.687, E3 +273479.356}
SPL {X  -163.980, Y  +355.035, Z    +0.000, E1   +53.657, E3 +273491.553}
SPL {X  -162.665, Y  +347.197, Z    +0.000, E1   +53.396, E3 +273504.816}
SPL {X  -161.218, Y  +340.437, Z    +0.000, E1   +53.207, E3 +273515.915}
SPL {X  -159.523, Y  +333.864, Z    +0.000, E1   +52.908, E3 +273527.537}
SPL {X  -157.624, Y  +327.563, Z    +0.000, E1   +52.705, E3 +273537.946}
SPL {X  -156.289, Y  +323.602, Z    +0.000, E1   +52.159, E3 +273546.835}
SPL {X  -153.877, Y  +317.168, Z    +0.000, E1   +51.945, E3 +273557.696}
SPL {X  -151.035, Y  +310.467, Z    +0.000, E1   +51.312, E3 +273570.942}
SPL {X  -139.567, Y  +289.276, Z    +0.000, E1   +56.334, E3 +273575.030}
SPL {X  -117.053, Y  +261.289, Z    +0.000, E1   +49.815, E3 +273688.564}
ENDSPLINE

SPLINE
SPL {X  -148.836, Y  +305.783, Z    +0.000, E1   +38.029, E3 +273780.041}
SPL {X  -161.816, Y  +343.065, Z    +0.000, E1   +22.147, E3 +273770.691}
SPL {X  -164.614, Y  +360.007, Z    +0.000, E1   +13.213, E3 +273766.478}
SPL {X  -165.520, Y  +371.933, Z    +0.000, E1    +6.276, E3 +273769.232}
SPL {X  -165.650, Y  +380.164, Z    +0.000, E1    +0.707, E3 +273767.701}
SPL {X  -165.650, Y  +384.850, Z    +0.000, E1    -3.598, E3 +273766.809}
SPL {X  -165.650, Y  +391.255, Z    +0.000, E1   -11.346, E3 +273765.150}
SPL {X  -165.650, Y  +398.038, Z    +0.000, E1   -20.113, E3 +273766.117}
SPL {X  -165.650, Y  +403.005, Z    +0.000, E1   -26.762, E3 +273765.299}
SPL {X  -165.650, Y  +415.469, Z    +0.000, E1   -43.461, E3 +273760.122}
SPL {X  -165.650, Y  +460.095, Z    +0.000, E1   -60.221, E3 +273778.383}
SPL {X  -165.650, Y  +535.749, Z    +0.000, E1   -60.559, E3 +273849.227}
ENDSPLINE

SPLINE
SPL {X  -165.650, Y  +516.750, Z    +0.000, E1   -54.244, E3 +273865.077}
ENDSPLINE

SPLINE
SPL {X  -165.650, Y  +524.345, Z    +0.000, E1   -54.115, E3 +273876.974}
SPL {X  -165.650, Y  +531.171, Z    +0.000, E1   -54.075, E3 +273887.413}
SPL {X  -165.650, Y  +538.771, Z    +0.000, E1   -53.840, E3 +273900.153}
SPL {X  -165.650, Y  +548.103, Z    +0.000, E1   -53.944, E3 +273913.500}
SPL {X  -165.650, Y  +558.071, Z    +0.000, E1   -53.870, E3 +273928.840}
SPL {X  -165.650, Y  +568.053, Z    +0.000, E1   -54.124, E3 +273942.018}
SPL {X  -165.650, Y  +577.021, Z    +0.000, E1   -53.813, E3 +273957.517}
SPL {X  -165.650, Y  +587.996, Z    +0.000, E1   -53.969, E3 +273972.754}
SPL {X  -165.650, Y  +595.185, Z    +0.000, E1   -53.962, E3 +273983.464}
SPL {X  -165.650, Y  +602.138, Z    +0.000, E1   -53.941, E3 +273993.958}
SPL {X  -165.650, Y  +610.307, Z    +0.000, E1   -53.995, E3 +274005.806}
SPL {X  -165.650, Y  +617.878, Z    +0.000, E1   -53.838, E3 +274018.062}
SPL {X  -165.650, Y  +626.374, Z    +0.000, E1   -54.092, E3 +274029.078}
SPL {X  -165.650, Y  +632.964, Z    +0.000, E1   -53.887, E3 +274040.205}
SPL {X  -165.650, Y  +640.262, Z    +0.000, E1   -53.965, E3 +274050.520}
SPL {X  -165.650, Y  +647.911, Z    +0.000, E1   -53.930, E3 +274062.274}
SPL {X  -165.650, Y  +656.836, Z    +0.000, E1   -54.184, E3 +274073.806}
SPL {X  -165.650, Y  +659.513, Z    +0.000, E1   -53.578, E3 +274081.536}
SPL {X  -165.650, Y  +667.820, Z    +0.000, E1   -53.975, E3 +274091.601}
SPL {X  -165.623, Y  +678.503, Z    +0.000, E1   -53.932, E3 +274107.953}
SPL {X  -165.171, Y  +688.090, Z    +0.000, E1   -54.025, E3 +274121.400}
SPL {X  -164.558, Y  +694.489, Z    +0.000, E1   -53.745, E3 +274132.750}
SPL {X  -163.580, Y  +701.606, Z    +0.000, E1   -53.591, E3 +274144.183}
SPL {X  -162.702, Y  +706.614, Z    +0.000, E1   -53.230, E3 +274153.849}
SPL {X  -160.941, Y  +714.715, Z    +0.000, E1   -53.321, E3 +274165.469}
SPL {X  -159.638, Y  +719.723, Z    +0.000, E1   -52.685, E3 +274176.471}
SPL {X  -157.868, Y  +725.674, Z    +0.000, E1   -52.862, E3 +274184.328}
SPL {X  -156.314, Y  +730.327, Z    +0.000, E1   -52.199, E3 +274195.010}
SPL {X  -153.975, Y  +736.588, Z    +0.000, E1   -51.877, E3 +274206.040}
SPL {X  -151.949, Y  +741.465, Z    +0.000, E1   -51.645, E3 +274214.445}
SPL {X  -149.075, Y  +747.727, Z    +0.000, E1   -52.134, E3 +274221.160}
SPL {X  -137.775, Y  +767.467, Z    +0.000, E1   -56.912, E3 +274223.823}
SPL {X  -128.847, Y  +779.607, Z    +0.000, E1   -49.118, E3 +274298.840}
SPL {X   -94.133, Y  +811.804, Z    +0.000, E1   -53.019, E3 +274353.474}
ENDSPLINE

SPLINE
SPL {X  -123.886, Y  +785.464, Z    +0.000, E1   -49.465, E3 +274438.500}
SPL {X  -152.385, Y  +740.452, Z    +0.000, E1   -34.821, E3 +274419.477}
SPL {X  -162.077, Y  +709.719, Z    +0.000, E1   -21.590, E3 +274421.324}
SPL {X  -164.499, Y  +694.994, Z    +0.000, E1   -13.860, E3 +274422.108}
SPL {X  -165.513, Y  +682.236, Z    +0.000, E1    -6.385, E3 +274420.444}
SPL {X  -165.650, Y  +675.776, Z    +0.000, E1    -2.014, E3 +274419.752}
SPL {X  -165.650, Y  +672.041, Z    +0.000, E1    +0.844, E3 +274418.700}
SPL {X  -165.650, Y  +667.328, Z    +0.000, E1    +5.806, E3 +274418.076}
SPL {X  -165.650, Y  +661.774, Z    +0.000, E1   +13.006, E3 +274416.400}
SPL {X  -165.650, Y  +654.085, Z    +0.000, E1   +23.232, E3 +274416.260}
SPL {X  -165.650, Y  +639.700, Z    +0.000, E1   +43.326, E3 +274410.387}
SPL {X  -165.650, Y  +605.320, Z    +0.000, E1   +76.562, E3 +274389.796}
SPL {X  -165.650, Y  +597.745, Z    +0.000, E1   +59.636, E3 +274427.798}
SPL {X  -165.650, Y  +596.360, Z    +0.000, E1   +54.978, E3 +274441.406}
SPL {X  -165.650, Y  +524.050, Z    +0.000, E1   +59.300, E3 +274503.312}
ENDSPLINE

SPLINE
SPL {X  -165.650, Y  +539.856, Z    +0.000, E1   +53.398, E3 +274518.959}
ENDSPLINE

SPLINE
SPL {X  -165.650, Y  +532.042, Z    +0.000, E1   +53.611, E3 +274529.430}
SPL {X  -165.650, Y  +523.239, Z    +0.000, E1   +53.520, E3 +274543.526}
SPL {X  -165.650, Y  +515.134, Z    +0.000, E1   +53.252, E3 +274557.255}
SPL {X  -165.650, Y  +505.685, Z    +0.000, E1   +53.701, E3 +274568.863}
SPL {X  -165.650, Y  +498.275, Z    +0.000, E1   +53.357, E3 +274582.170}
SPL {X  -165.650, Y  +491.031, Z    +0.000, E1   +53.348, E3 +274593.190}
SPL {X  -165.650, Y  +479.077, Z    +0.000, E1   +55.039, E3 +274600.313}
SPL {X  -165.650, Y  +450.615, Z    +0.000, E1   +59.721, E3 +274606.819}
SPL {X  -165.650, Y  +449.326, Z    +0.000, E1   +58.606, E3 +274615.868}
SPL {X  -165.650, Y  +442.154, Z    +0.000, E1   +58.369, E3 +274626.492}
SPL {X  -165.650, Y  +437.405, Z    +0.000, E1   +57.663, E3 +274637.102}
SPL {X  -165.650, Y  +432.227, Z    +0.000, E1   +57.103, E3 +274647.590}
SPL {X  -165.650, Y  +428.683, Z    +0.000, E1   +56.222, E3 +274657.944}
SPL {X  -165.650, Y  +424.202, Z    +0.000, E1   +55.382, E3 +274669.633}
SPL {X  -165.650, Y  +418.469, Z    +0.000, E1   +54.594, E3 +274682.741}
SPL {X  -165.650, Y  +413.857, Z    +0.000, E1   +53.683, E3 +274695.312}
SPL {X  -165.650, Y  +405.379, Z    +0.000, E1   +53.922, E3 +274706.426}
SPL {X  -165.650, Y  +400.791, Z    +0.000, E1   +53.827, E3 +274713.840}
SPL {X  -165.650, Y  +393.046, Z    +0.000, E1   +53.951, E3 +274724.732}
SPL {X  -165.650, Y  +383.306, Z    +0.000, E1   +53.987, E3 +274739.010}
SPL {X  -165.640, Y  +376.676, Z    +0.000, E1   +53.760, E3 +274750.176}
SPL {X  -165.408, Y  +369.556, Z    +0.000, E1   +53.942, E3 +274759.727}
SPL {X  -164.927, Y  +363.041, Z    +0.000, E1   +53.687, E3 +274771.023}
SPL {X  -164.096, Y  +355.862, Z    +0.000, E1   +53.838, E3 +274780.753}
SPL {X  -163.142, Y  +349.785, Z    +0.000, E1   +53.493, E3 +274791.969}
SPL {X  -161.604, Y  +342.113, Z    +0.000, E1   +53.155, E3 +274805.463}
SPL {X  -160.424, Y  +337.221, Z    +0.000, E1   +52.694, E3 +274815.303}
SPL {X  -158.192, Y  +329.354, Z    +0.000, E1   +52.890, E3 +274826.135}
SPL {X  -156.289, Y  +323.602, Z    +0.000, E1   +52.159, E3 +274838.502}
SPL {X  -154.898, Y  +319.792, Z    +0.000, E1   +51.850, E3 +274845.837}
SPL {X  -152.682, Y  +314.249, Z    +0.000, E1   +51.841, E3 +274854.234}
SPL {X  -150.607, Y  +309.525, Z    +0.000, E1   +51.147, E3 +274864.719}
SPL {X  -139.567, Y  +289.276, Z    +0.000, E1   +56.334, E3 +274866.697}
SPL {X  -117.053, Y  +261.289, Z    +0.000, E1   +49.815, E3 +274980.230}
ENDSPLINE

SPLINE
SPL {X  -148.836, Y  +305.783, Z    +0.000, E1   +38.029, E3 +275071.708}
SPL {X  -161.816, Y  +343.065, Z    +0.000, E1   +22.147, E3 +275062.358}
SPL {X  -164.614, Y  +360.007, Z    +0.000, E1   +13.213, E3 +275058.144}
SPL {X  -165.520, Y  +371.933, Z    +0.000, E1    +6.276, E3 +275060.899}
SPL {X  -165.650, Y  +378.704, Z    +0.000, E1    +1.700, E3 +275059.768}
SPL {X  -165.650, Y  +382.197, Z    +0.000, E1    -1.038, E3 +275058.841}
SPL {X  -165.650, Y  +386.782, Z    +0.000, E1    -5.783, E3 +275058.319}
SPL {X  -165.650, Y  +392.406, Z    +0.000, E1   -13.042, E3 +275056.216}
SPL {X  -165.650, Y  +398.038, Z    +0.000, E1   -20.113, E3 +275057.784}
SPL {X  -165.650, Y  +403.005, Z    +0.000, E1   -26.762, E3 +275056.966}
SPL {X  -165.650, Y  +415.469, Z    +0.000, E1   -43.461, E3 +275051.789}
SPL {X  -165.650, Y  +460.095, Z    +0.000, E1   -60.221, E3 +275070.050}
SPL {X  -165.650, Y  +537.366, Z    +0.000, E1   -61.810, E3 +275134.626}
ENDSPLINE

SPLINE
SPL {X  -165.650, Y  +520.647, Z    +0.000, E1   -55.836, E3 +275152.318}
ENDSPLINE

SPLINE
SPL {X  -165.650, Y  +521.328, Z    +0.000, E1   -53.870, E3 +275165.735}
SPL {X  -165.650, Y  +531.171, Z    +0.000, E1   -54.075, E3 +275179.079}
SPL {X  -165.650, Y  +538.771, Z    +0.000, E1   -53.840, E3 +275191.820}
SPL {X  -165.650, Y  +548.103, Z    +0.000, E1   -53.944, E3 +275205.166}
SPL {X  -165.650, Y  +558.071, Z    +0.000, E1   -53.870, E3 +275220.507}
SPL {X  -165.650, Y  +568.053, Z    +0.000, E1   -54.124, E3 +275233.685}
SPL {X  -165.650, Y  +574.396, Z    +0.000, E1   -53.807, E3 +275245.076}
SPL {X  -165.650, Y  +579.991, Z    +0.000, E1   -53.716, E3 +275253.986}
SPL {X  -165.650, Y  +587.996, Z    +0.000, E1   -53.969, E3 +275264.421}
SPL {X  -165.650, Y  +595.185, Z    +0.000, E1   -53.962, E3 +275275.130}
SPL {X  -165.650, Y  +602.138, Z    +0.000, E1   -53.941, E3 +275285.625}
SPL {X  -165.650, Y  +610.307, Z    +0.000, E1   -53.995, E3 +275297.472}
SPL {X  -165.650, Y  +617.878, Z    +0.000, E1   -53.838, E3 +275309.729}
SPL {X  -165.650, Y  +626.374, Z    +0.000, E1   -54.092, E3 +275320.744}
SPL {X  -165.650, Y  +632.964, Z    +0.000, E1   -53.887, E3 +275331.872}
SPL {X  -165.650, Y  +640.262, Z    +0.000, E1   -53.965, E3 +275342.187}
SPL {X  -165.650, Y  +647.911, Z    +0.000, E1   -53.930, E3 +275353.941}
SPL {X  -165.650, Y  +656.836, Z    +0.000, E1   -54.184, E3 +275365.473}
SPL {X  -165.650, Y  +659.513, Z    +0.000, E1   -53.578, E3 +275373.203}
SPL {X  -165.650, Y  +667.820, Z    +0.000, E1   -53.975, E3 +275383.268}
SPL {X  -165.623, Y  +678.503, Z    +0.000, E1   -53.932, E3 +275399.619}
SPL {X  -165.027, Y  +689.850, Z    +0.000, E1   -53.862, E3 +275416.883}
SPL {X  -163.840, Y  +699.919, Z    +0.000, E1   -53.732, E3 +275432.665}
SPL {X  -162.702, Y  +706.614, Z    +0.000, E1   -53.230, E3 +275445.516}
SPL {X  -161.265, Y  +713.361, Z    +0.000, E1   -53.436, E3 +275454.325}
SPL {X  -159.936, Y  +718.632, Z    +0.000, E1   -52.857, E3 +275465.654}
SPL {X  -157.868, Y  +725.674, Z    +0.000, E1   -52.862, E3 +275475.995}
SPL {X  -156.314, Y  +730.327, Z    +0.000, E1   -52.199, E3 +275486.676}
SPL {X  -153.975, Y  +736.588, Z    +0.000, E1   -51.877, E3 +275497.707}
SPL {X  -151.949, Y  +741.465, Z    +0.000, E1   -51.645, E3 +275506.112}
SPL {X  -149.075, Y  +747.727, Z    +0.000, E1   -52.134, E3 +275512.827}
SPL {X  -137.775, Y  +767.467, Z    +0.000, E1   -56.912, E3 +275515.490}
SPL {X  -128.847, Y  +779.607, Z    +0.000, E1   -49.118, E3 +275590.506}
SPL {X   -94.133, Y  +811.804, Z    +0.000, E1   -53.019, E3 +275645.141}
ENDSPLINE

SPLINE
SPL {X  -134.098, Y  +772.750, Z    +0.000, E1   -45.587, E3 +275720.435}
SPL {X  -155.319, Y  +733.085, Z    +0.000, E1   -31.947, E3 +275711.313}
SPL {X  -162.077, Y  +709.719, Z    +0.000, E1   -21.590, E3 +275712.990}
SPL {X  -164.499, Y  +694.994, Z    +0.000, E1   -13.860, E3 +275713.775}
SPL {X  -165.513, Y  +682.236, Z    +0.000, E1    -6.385, E3 +275712.111}
SPL {X  -165.650, Y  +675.776, Z    +0.000, E1    -2.014, E3 +275711.418}
SPL {X  -165.650, Y  +672.938, Z    +0.000, E1    +0.157, E3 +275710.434}
SPL {X  -165.650, Y  +669.402, Z    +0.000, E1    +3.448, E3 +275709.825}
SPL {X  -165.650, Y  +663.061, Z    +0.000, E1   +11.076, E3 +275708.819}
SPL {X  -165.650, Y  +656.573, Z    +0.000, E1   +19.875, E3 +275708.626}
SPL {X  -165.650, Y  +650.769, Z    +0.000, E1   +28.083, E3 +275706.992}
SPL {X  -165.650, Y  +639.700, Z    +0.000, E1   +43.326, E3 +275702.054}
SPL {X  -165.650, Y  +605.320, Z    +0.000, E1   +76.562, E3 +275681.463}
SPL {X  -165.650, Y  +597.745, Z    +0.000, E1   +59.636, E3 +275719.464}
SPL {X  -165.650, Y  +596.360, Z    +0.000, E1   +54.978, E3 +275733.072}
SPL {X  -165.650, Y  +521.429, Z    +0.000, E1   +61.144, E3 +275786.303}
ENDSPLINE

SPLINE
SPL {X  -165.650, Y  +526.028, Z    +0.000, E1   +58.071, E3 +275800.078}
SPL {X  -165.650, Y  +539.856, Z    +0.000, E1   +53.398, E3 +275810.626}
ENDSPLINE

SPLINE
SPL {X  -165.650, Y  +532.042, Z    +0.000, E1   +53.611, E3 +275821.097}
SPL {X  -165.650, Y  +526.147, Z    +0.000, E1   +53.495, E3 +275830.736}
SPL {X  -165.650, Y  +517.365, Z    +0.000, E1   +53.387, E3 +275844.904}
SPL {X  -165.650, Y  +505.685, Z    +0.000, E1   +53.701, E3 +275860.529}
SPL {X  -165.650, Y  +498.275, Z    +0.000, E1   +53.357, E3 +275873.837}
SPL {X  -165.650, Y  +487.031, Z    +0.000, E1   +53.931, E3 +275887.246}
SPL {X  -165.650, Y  +450.615, Z    +0.000, E1   +59.721, E3 +275898.486}
SPL {X  -165.650, Y  +449.326, Z    +0.000, E1   +58.606, E3 +275907.535}
SPL {X  -165.650, Y  +442.154, Z    +0.000, E1   +58.369, E3 +275918.159}
SPL {X  -165.650, Y  +437.405, Z    +0.000, E1   +57.663, E3 +275928.769}
SPL {X  -165.650, Y  +432.227, Z    +0.000, E1   +57.103, E3 +275939.256}
SPL {X  -165.650, Y  +428.683, Z    +0.000, E1   +56.222, E3 +275949.611}
SPL {X  -165.650, Y  +424.202, Z    +0.000, E1   +55.382, E3 +275961.300}
SPL {X  -165.650, Y  +418.756, Z    +0.000, E1   +54.154, E3 +275976.979}
SPL {X  -165.650, Y  +410.508, Z    +0.000, E1   +54.007, E3 +275989.934}
SPL {X  -165.650, Y  +403.104, Z    +0.000, E1   +53.908, E3 +276001.716}
SPL {X  -165.650, Y  +393.046, Z    +0.000, E1   +53.951, E3 +276016.399}
SPL {X  -165.650, Y  +383.306, Z    +0.000, E1   +53.987, E3 +276030.676}
SPL {X  -165.640, Y  +376.676, Z    +0.000, E1   +53.760, E3 +276041.843}
SPL {X  -165.408, Y  +369.556, Z    +0.000, E1   +53.942, E3 +276051.394}
SPL {X  -164.927, Y  +363.041, Z    +0.000, E1   +53.687, E3 +276062.690}
SPL {X  -163.980, Y  +355.035, Z    +0.000, E1   +53.657, E3 +276074.886}
SPL {X  -162.665, Y  +347.197, Z    +0.000, E1   +53.396, E3 +276088.149}
SPL {X  -161.218, Y  +340.437, Z    +0.000, E1   +53.207, E3 +276099.248}
SPL {X  -159.523, Y  +333.864, Z    +0.000, E1   +52.908, E3 +276110.870}
SPL {X  -157.624, Y  +327.563, Z    +0.000, E1   +52.705, E3 +276121.280}
SPL {X  -156.289, Y  +323.602, Z    +0.000, E1   +52.159, E3 +276130.168}
SPL {X  -153.877, Y  +317.168, Z    +0.000, E1   +51.945, E3 +276141.030}
SPL {X  -151.035, Y  +310.467, Z    +0.000, E1   +51.312, E3 +276154.275}
SPL {X  -139.567, Y  +289.276, Z    +0.000, E1   +56.334, E3 +276158.363}
SPL {X  -117.053, Y  +261.289, Z    +0.000, E1   +49.815, E3 +276271.897}
ENDSPLINE

SPLINE
SPL {X  -148.836, Y  +305.783, Z    +0.000, E1   +38.029, E3 +276363.375}
SPL {X  -161.816, Y  +343.065, Z    +0.000, E1   +22.147, E3 +276354.025}
SPL {X  -164.614, Y  +360.007, Z    +0.000, E1   +13.213, E3 +276349.811}
SPL {X  -165.520, Y  +371.933, Z    +0.000, E1    +6.276, E3 +276352.565}
SPL {X  -165.650, Y  +378.704, Z    +0.000, E1    +1.700, E3 +276351.435}
SPL {X  -165.650, Y  +382.197, Z    +0.000, E1    -1.038, E3 +276350.508}
SPL {X  -165.650, Y  +386.782, Z    +0.000, E1    -5.783, E3 +276349.986}
SPL {X  -165.650, Y  +392.406, Z    +0.000, E1   -13.042, E3 +276347.883}
SPL {X  -165.650, Y  +400.489, Z    +0.000, E1   -23.243, E3 +276349.047}
SPL {X  -165.650, Y  +415.469, Z    +0.000, E1   -43.461, E3 +276343.455}
SPL {X  -165.650, Y  +460.095, Z    +0.000, E1   -60.221, E3 +276361.717}
SPL {X  -165.650, Y  +535.749, Z    +0.000, E1   -60.559, E3 +276432.560}
ENDSPLINE

SPLINE
SPL {X  -165.650, Y  +516.866, Z    +0.000, E1   -54.768, E3 +276445.110}
ENDSPLINE

SPLINE
SPL {X  -165.650, Y  +521.328, Z    +0.000, E1   -53.870, E3 +276457.402}
SPL {X  -165.650, Y  +531.171, Z    +0.000, E1   -54.075, E3 +276470.746}
SPL {X  -165.650, Y  +538.771, Z    +0.000, E1   -53.840, E3 +276483.486}
SPL {X  -165.650, Y  +548.103, Z    +0.000, E1   -53.944, E3 +276496.833}
SPL {X  -165.650, Y  +558.071, Z    +0.000, E1   -53.870, E3 +276512.174}
SPL {X  -165.650, Y  +568.053, Z    +0.000, E1   -54.124, E3 +276525.351}
SPL {X  -165.650, Y  +577.021, Z    +0.000, E1   -53.813, E3 +276540.850}
SPL {X  -165.650, Y  +587.996, Z    +0.000, E1   -53.969, E3 +276556.088}
SPL {X  -165.650, Y  +595.185, Z    +0.000, E1   -53.962, E3 +276566.797}
SPL {X  -165.650, Y  +602.138, Z    +0.000, E1   -53.941, E3 +276577.291}
SPL {X  -165.650, Y  +610.307, Z    +0.000, E1   -53.995, E3 +276589.139}
SPL {X  -165.650, Y  +617.878, Z    +0.000, E1   -53.838, E3 +276601.396}
SPL {X  -165.650, Y  +627.853, Z    +0.000, E1   -53.937, E3 +276615.749}
SPL {X  -165.650, Y  +638.510, Z    +0.000, E1   -54.057, E3 +276630.809}
SPL {X  -165.650, Y  +647.911, Z    +0.000, E1   -53.930, E3 +276645.608}
SPL {X  -165.650, Y  +658.189, Z    +0.000, E1   -53.932, E3 +276660.908}
SPL {X  -165.650, Y  +667.820, Z    +0.000, E1   -53.975, E3 +276674.934}
SPL {X  -165.623, Y  +678.503, Z    +0.000, E1   -53.932, E3 +276691.286}
SPL {X  -165.171, Y  +688.090, Z    +0.000, E1   -54.025, E3 +276704.734}
SPL {X  -164.558, Y  +694.489, Z    +0.000, E1   -53.745, E3 +276716.083}
SPL {X  -163.580, Y  +701.606, Z    +0.000, E1   -53.591, E3 +276727.516}
SPL {X  -162.702, Y  +706.614, Z    +0.000, E1   -53.230, E3 +276737.183}
SPL {X  -160.941, Y  +714.715, Z    +0.000, E1   -53.321, E3 +276748.802}
SPL {X  -159.638, Y  +719.723, Z    +0.000, E1   -52.685, E3 +276759.805}
SPL {X  -157.521, Y  +726.754, Z    +0.000, E1   -52.585, E3 +276771.000}
SPL {X  -155.632, Y  +732.234, Z    +0.000, E1   -52.209, E3 +276781.047}
SPL {X  -153.975, Y  +736.588, Z    +0.000, E1   -51.877, E3 +276789.373}
SPL {X  -151.949, Y  +741.465, Z    +0.000, E1   -51.645, E3 +276797.779}
SPL {X  -149.075, Y  +747.727, Z    +0.000, E1   -52.134, E3 +276804.493}
SPL {X  -137.775, Y  +767.467, Z    +0.000, E1   -56.912, E3 +276807.157}
SPL {X  -128.847, Y  +779.607, Z    +0.000, E1   -49.118, E3 +276882.173}
SPL {X   -94.133, Y  +811.804, Z    +0.000, E1   -53.019, E3 +276936.807}
ENDSPLINE

SPLINE
SPL {X  -134.098, Y  +772.750, Z    +0.000, E1   -45.587, E3 +277012.102}
SPL {X  -155.319, Y  +733.085, Z    +0.000, E1   -31.947, E3 +277002.979}
SPL {X  -162.077, Y  +709.719, Z    +0.000, E1   -21.590, E3 +277004.657}
SPL {X  -164.499, Y  +694.994, Z    +0.000, E1   -13.860, E3 +277005.442}
SPL {X  -165.382, Y  +684.927, Z    +0.000, E1    -7.984, E3 +277003.619}
SPL {X  -165.645, Y  +676.778, Z    +0.000, E1    -2.777, E3 +277003.341}
SPL {X  -165.650, Y  +672.041, Z    +0.000, E1    +0.844, E3 +277002.033}
SPL {X  -165.650, Y  +667.328, Z    +0.000, E1    +5.806, E3 +277001.410}
SPL {X  -165.650, Y  +661.774, Z    +0.000, E1   +13.006, E3 +276999.734}
SPL {X  -165.650, Y  +656.573, Z    +0.000, E1   +19.875, E3 +277000.292}
SPL {X  -165.650, Y  +647.335, Z    +0.000, E1   +32.835, E3 +276997.214}
SPL {X  -165.650, Y  +637.438, Z    +0.000, E1   +46.409, E3 +276992.574}
SPL {X  -165.650, Y  +605.320, Z    +0.000, E1   +76.562, E3 +276973.130}
SPL {X  -165.650, Y  +596.505, Z    +0.000, E1   +55.802, E3 +277022.485}
SPL {X  -165.650, Y  +524.050, Z    +0.000, E1   +59.300, E3 +277086.645}
ENDSPLINE

SPLINE
SPL {X  -165.650, Y  +539.856, Z    +0.000, E1   +53.398, E3 +277102.292}
ENDSPLINE

SPLINE
SPL {X  -165.650, Y  +530.389, Z    +0.000, E1   +53.621, E3 +277115.298}
SPL {X  -165.650, Y  +521.849, Z    +0.000, E1   +53.452, E3 +277129.237}
SPL {X  -165.650, Y  +515.134, Z    +0.000, E1   +53.252, E3 +277140.588}
SPL {X  -165.650, Y  +505.685, Z    +0.000, E1   +53.701, E3 +277152.196}
SPL {X  -165.650, Y  +498.275, Z    +0.000, E1   +53.357, E3 +277165.504}
SPL {X  -165.650, Y  +491.031, Z    +0.000, E1   +53.348, E3 +277176.524}
SPL {X  -165.650, Y  +479.077, Z    +0.000, E1   +55.039, E3 +277183.647}
SPL {X  -165.650, Y  +450.615, Z    +0.000, E1   +59.721, E3 +277190.152}
SPL {X  -165.650, Y  +449.326, Z    +0.000, E1   +58.606, E3 +277199.202}
SPL {X  -165.650, Y  +442.154, Z    +0.000, E1   +58.369, E3 +277209.826}
SPL {X  -165.650, Y  +437.405, Z    +0.000, E1   +57.663, E3 +277220.435}
SPL {X  -165.650, Y  +432.227, Z    +0.000, E1   +57.103, E3 +277230.923}
SPL {X  -165.650, Y  +428.683, Z    +0.000, E1   +56.222, E3 +277241.277}
SPL {X  -165.650, Y  +424.202, Z    +0.000, E1   +55.382, E3 +277252.966}
SPL {X  -165.650, Y  +418.756, Z    +0.000, E1   +54.154, E3 +277268.645}
SPL {X  -165.650, Y  +407.872, Z    +0.000, E1   +54.003, E3 +277285.731}
SPL {X  -165.650, Y  +400.791, Z    +0.000, E1   +53.827, E3 +277297.173}
SPL {X  -165.650, Y  +393.046, Z    +0.000, E1   +53.951, E3 +277308.066}
SPL {X  -165.650, Y  +383.306, Z    +0.000, E1   +53.987, E3 +277322.343}
SPL {X  -165.640, Y  +376.676, Z    +0.000, E1   +53.760, E3 +277333.510}
SPL {X  -165.408, Y  +369.556, Z    +0.000, E1   +53.942, E3 +277343.061}
SPL {X  -164.927, Y  +363.041, Z    +0.000, E1   +53.687, E3 +277354.356}
SPL {X  -164.096, Y  +355.862, Z    +0.000, E1   +53.838, E3 +277364.087}
SPL {X  -162.936, Y  +348.637, Z    +0.000, E1   +53.390, E3 +277377.803}
SPL {X  -161.218, Y  +340.437, Z    +0.000, E1   +53.207, E3 +277390.915}
SPL {X  -159.523, Y  +333.864, Z    +0.000, E1   +52.908, E3 +277402.537}
SPL {X  -157.624, Y  +327.563, Z    +0.000, E1   +52.705, E3 +277412.946}
SPL {X  -155.665, Y  +321.859, Z    +0.000, E1   +52.064, E3 +277425.119}
SPL {X  -152.682, Y  +314.249, Z    +0.000, E1   +51.841, E3 +277437.567}
SPL {X  -150.607, Y  +309.525, Z    +0.000, E1   +51.147, E3 +277448.052}
SPL {X  -142.104, Y  +293.374, Z    +0.000, E1   +55.775, E3 +277447.784}
SPL {X  -134.755, Y  +282.163, Z    +0.000, E1   +57.236, E3 +277454.052}
SPL {X  -117.053, Y  +261.289, Z    +0.000, E1   +49.815, E3 +277563.564}
ENDSPLINE

SPLINE
SPL {X  -148.836, Y  +305.783, Z    +0.000, E1   +38.029, E3 +277655.041}
SPL {X  -161.816, Y  +343.065, Z    +0.000, E1   +22.147, E3 +277645.691}
SPL {X  -164.614, Y  +360.007, Z    +0.000, E1   +13.213, E3 +277641.478}
SPL {X  -165.520, Y  +371.933, Z    +0.000, E1    +6.276, E3 +277644.232}
SPL {X  -165.650, Y  +378.704, Z    +0.000, E1    +1.700, E3 +277643.101}
SPL {X  -165.650, Y  +382.197, Z    +0.000, E1    -1.038, E3 +277642.175}
SPL {X  -165.650, Y  +386.782, Z    +0.000, E1    -5.783, E3 +277641.652}
SPL {X  -165.650, Y  +392.406, Z    +0.000, E1   -13.042, E3 +277639.550}
SPL {X  -165.650, Y  +398.038, Z    +0.000, E1   -20.113, E3 +277641.117}
SPL {X  -165.650, Y  +403.005, Z    +0.000, E1   -26.762, E3 +277640.299}
SPL {X  -165.650, Y  +415.469, Z    +0.000, E1   -43.461, E3 +277635.122}
SPL {X  -165.650, Y  +460.095, Z    +0.000, E1   -60.221, E3 +277653.383}
SPL {X  -165.650, Y  +535.749, Z    +0.000, E1   -60.559, E3 +277724.227}
ENDSPLINE

SPLINE
SPL {X  -165.650, Y  +516.750, Z    +0.000, E1   -54.244, E3 +277740.077}
ENDSPLINE

SPLINE
SPL {X  -165.650, Y  +524.345, Z    +0.000, E1   -54.115, E3 +277751.974}
SPL {X  -165.650, Y  +531.171, Z    +0.000, E1   -54.075, E3 +277762.413}
SPL {X  -165.650, Y  +538.771, Z    +0.000, E1   -53.840, E3 +277775.153}
SPL {X  -165.650, Y  +545.884, Z    +0.000, E1   -53.883, E3 +277785.458}
SPL {X  -165.650, Y  +553.081, Z    +0.000, E1   -53.834, E3 +277796.591}
SPL {X  -165.650, Y  +560.989, Z    +0.000, E1   -53.974, E3 +277807.428}
SPL {X  -165.650, Y  +568.053, Z    +0.000, E1   -54.124, E3 +277817.018}
SPL {X  -165.650, Y  +577.021, Z    +0.000, E1   -53.813, E3 +277832.517}
SPL {X  -165.650, Y  +587.996, Z    +0.000, E1   -53.969, E3 +277847.754}
SPL {X  -165.650, Y  +595.185, Z    +0.000, E1   -53.962, E3 +277858.464}
SPL {X  -165.650, Y  +602.138, Z    +0.000, E1   -53.941, E3 +277868.958}
SPL {X  -165.650, Y  +610.307, Z    +0.000, E1   -53.995, E3 +277880.806}
SPL {X  -165.650, Y  +617.878, Z    +0.000, E1   -53.838, E3 +277893.062}
SPL {X  -165.650, Y  +626.374, Z    +0.000, E1   -54.092, E3 +277904.078}
SPL {X  -165.650, Y  +632.964, Z    +0.000, E1   -53.887, E3 +277915.205}
SPL {X  -165.650, Y  +643.032, Z    +0.000, E1   -53.946, E3 +277929.950}
SPL {X  -165.650, Y  +654.069, Z    +0.000, E1   -54.108, E3 +277945.309}
SPL {X  -165.650, Y  +659.513, Z    +0.000, E1   -53.578, E3 +277956.536}
SPL {X  -165.650, Y  +667.820, Z    +0.000, E1   -53.975, E3 +277966.601}
SPL {X  -165.650, Y  +674.957, Z    +0.000, E1   -53.977, E3 +277977.113}
SPL {X  -165.574, Y  +680.515, Z    +0.000, E1   -53.820, E3 +277986.440}
SPL {X  -165.171, Y  +688.090, Z    +0.000, E1   -54.025, E3 +277996.400}
SPL {X  -164.558, Y  +694.489, Z    +0.000, E1   -53.745, E3 +278007.750}
SPL {X  -163.580, Y  +701.606, Z    +0.000, E1   -53.591, E3 +278019.183}
SPL {X  -162.702, Y  +706.614, Z    +0.000, E1   -53.230, E3 +278028.849}
SPL {X  -161.265, Y  +713.361, Z    +0.000, E1   -53.436, E3 +278037.658}
SPL {X  -159.936, Y  +718.632, Z    +0.000, E1   -52.857, E3 +278048.987}
SPL {X  -157.868, Y  +725.674, Z    +0.000, E1   -52.862, E3 +278059.328}
SPL {X  -156.314, Y  +730.327, Z    +0.000, E1   -52.199, E3 +278070.010}
SPL {X  -153.975, Y  +736.588, Z    +0.000, E1   -51.877, E3 +278081.040}
SPL {X  -151.181, Y  +743.207, Z    +0.000, E1   -51.549, E3 +278092.661}
SPL {X  -146.528, Y  +752.763, Z    +0.000, E1   -53.481, E3 +278096.838}
SPL {X  -137.775, Y  +767.467, Z    +0.000, E1   -56.912, E3 +278098.823}
SPL {X  -128.847, Y  +779.607, Z    +0.000, E1   -49.118, E3 +278173.840}
SPL {X   -94.133, Y  +811.804, Z    +0.000, E1   -53.019, E3 +278228.474}
ENDSPLINE

SPLINE
SPL {X  -134.098, Y  +772.750, Z    +0.000, E1   -45.587, E3 +278303.768}
SPL {X  -155.319, Y  +733.085, Z    +0.000, E1   -31.947, E3 +278294.646}
SPL {X  -162.077, Y  +709.719, Z    +0.000, E1   -21.590, E3 +278296.324}
SPL {X  -164.499, Y  +694.994, Z    +0.000, E1   -13.860, E3 +278297.108}
SPL {X  -165.382, Y  +684.927, Z    +0.000, E1    -7.984, E3 +278295.286}
SPL {X  -165.645, Y  +676.778, Z    +0.000, E1    -2.777, E3 +278295.008}
SPL {X  -165.650, Y  +672.938, Z    +0.000, E1    +0.157, E3 +278293.767}
SPL {X  -165.650, Y  +669.402, Z    +0.000, E1    +3.448, E3 +278293.158}
SPL {X  -165.650, Y  +663.061, Z    +0.000, E1   +11.076, E3 +278292.152}
SPL {X  -165.650, Y  +654.085, Z    +0.000, E1   +23.232, E3 +278291.260}
SPL {X  -165.650, Y  +639.700, Z    +0.000, E1   +43.326, E3 +278285.387}
SPL {X  -165.650, Y  +605.320, Z    +0.000, E1   +76.562, E3 +278264.796}
SPL {X  -165.650, Y  +596.505, Z    +0.000, E1   +55.802, E3 +278314.152}
SPL {X  -165.650, Y  +524.050, Z    +0.000, E1   +59.300, E3 +278378.312}
ENDSPLINE

SPLINE
SPL {X  -165.650, Y  +539.856, Z    +0.000, E1   +53.398, E3 +278393.959}
ENDSPLINE

SPLINE
SPL {X  -165.650, Y  +532.042, Z    +0.000, E1   +53.611, E3 +278404.430}
SPL {X  -165.650, Y  +523.239, Z    +0.000, E1   +53.520, E3 +278418.526}
SPL {X  -165.650, Y  +512.447, Z    +0.000, E1   +53.456, E3 +278435.163}
SPL {X  -165.650, Y  +503.994, Z    +0.000, E1   +53.652, E3 +278446.602}
SPL {X  -165.650, Y  +498.275, Z    +0.000, E1   +53.357, E3 +278457.170}
SPL {X  -165.650, Y  +487.031, Z    +0.000, E1   +53.931, E3 +278470.579}
SPL {X  -165.650, Y  +450.615, Z    +0.000, E1   +59.721, E3 +278481.819}
SPL {X  -165.650, Y  +449.326, Z    +0.000, E1   +58.606, E3 +278490.868}
SPL {X  -165.650, Y  +442.154, Z    +0.000, E1   +58.369, E3 +278501.492}
SPL {X  -165.650, Y  +437.405, Z    +0.000, E1   +57.663, E3 +278512.102}
SPL {X  -165.650, Y  +432.227, Z    +0.000, E1   +57.103, E3 +278522.590}
SPL {X  -165.650, Y  +428.683, Z    +0.000, E1   +56.222, E3 +278532.944}
SPL {X  -165.650, Y  +424.202, Z    +0.000, E1   +55.382, E3 +278544.633}
SPL {X  -165.650, Y  +418.756, Z    +0.000, E1   +54.154, E3 +278560.312}
SPL {X  -165.650, Y  +410.508, Z    +0.000, E1   +54.007, E3 +278573.267}
SPL {X  -165.650, Y  +403.104, Z    +0.000, E1   +53.908, E3 +278585.049}
SPL {X  -165.650, Y  +391.401, Z    +0.000, E1   +53.934, E3 +278602.440}
SPL {X  -165.650, Y  +378.987, Z    +0.000, E1   +53.974, E3 +278620.636}
SPL {X  -165.408, Y  +369.556, Z    +0.000, E1   +53.942, E3 +278634.727}
SPL {X  -164.927, Y  +363.041, Z    +0.000, E1   +53.687, E3 +278646.023}
SPL {X  -164.096, Y  +355.862, Z    +0.000, E1   +53.838, E3 +278655.753}
SPL {X  -163.142, Y  +349.785, Z    +0.000, E1   +53.493, E3 +278666.969}
SPL {X  -161.604, Y  +342.113, Z    +0.000, E1   +53.155, E3 +278680.463}
SPL {X  -160.424, Y  +337.221, Z    +0.000, E1   +52.694, E3 +278690.303}
SPL {X  -158.192, Y  +329.354, Z    +0.000, E1   +52.890, E3 +278701.135}
SPL {X  -156.289, Y  +323.602, Z    +0.000, E1   +52.159, E3 +278713.502}
SPL {X  -154.898, Y  +319.792, Z    +0.000, E1   +51.850, E3 +278720.837}
SPL {X  -152.682, Y  +314.249, Z    +0.000, E1   +51.841, E3 +278729.234}
SPL {X  -150.607, Y  +309.525, Z    +0.000, E1   +51.147, E3 +278739.719}
SPL {X  -139.567, Y  +289.276, Z    +0.000, E1   +56.334, E3 +278741.697}
SPL {X  -117.053, Y  +261.289, Z    +0.000, E1   +49.815, E3 +278855.230}
ENDSPLINE

SPLINE
SPL {X  -148.836, Y  +305.783, Z    +0.000, E1   +38.029, E3 +278946.708}
SPL {X  -161.816, Y  +343.065, Z    +0.000, E1   +22.147, E3 +278937.358}
SPL {X  -164.614, Y  +360.007, Z    +0.000, E1   +13.213, E3 +278933.144}
SPL {X  -165.520, Y  +371.933, Z    +0.000, E1    +6.276, E3 +278935.899}
SPL {X  -165.650, Y  +378.704, Z    +0.000, E1    +1.700, E3 +278934.768}
SPL {X  -165.650, Y  +382.197, Z    +0.000, E1    -1.038, E3 +278933.841}
SPL {X  -165.650, Y  +386.782, Z    +0.000, E1    -5.783, E3 +278933.319}
SPL {X  -165.650, Y  +392.406, Z    +0.000, E1   -13.042, E3 +278931.216}
SPL {X  -165.650, Y  +398.038, Z    +0.000, E1   -20.113, E3 +278932.784}
SPL {X  -165.650, Y  +403.005, Z    +0.000, E1   -26.762, E3 +278931.966}
SPL {X  -165.650, Y  +415.469, Z    +0.000, E1   -43.461, E3 +278926.789}
SPL {X  -165.650, Y  +460.095, Z    +0.000, E1   -60.221, E3 +278945.050}
SPL {X  -165.650, Y  +537.366, Z    +0.000, E1   -61.810, E3 +279009.626}
ENDSPLINE

SPLINE
SPL {X  -165.650, Y  +520.647, Z    +0.000, E1   -55.836, E3 +279027.318}
ENDSPLINE

SPLINE
SPL {X  -165.650, Y  +521.328, Z    +0.000, E1   -53.870, E3 +279040.735}
SPL {X  -165.650, Y  +531.171, Z    +0.000, E1   -54.075, E3 +279054.079}
SPL {X  -165.650, Y  +538.771, Z    +0.000, E1   -53.840, E3 +279066.820}
SPL {X  -165.650, Y  +548.103, Z    +0.000, E1   -53.944, E3 +279080.166}
SPL {X  -165.650, Y  +558.071, Z    +0.000, E1   -53.870, E3 +279095.507}
SPL {X  -165.650, Y  +568.053, Z    +0.000, E1   -54.124, E3 +279108.685}
SPL {X  -165.650, Y  +574.396, Z    +0.000, E1   -53.807, E3 +279120.076}
SPL {X  -165.650, Y  +579.991, Z    +0.000, E1   -53.716, E3 +279128.986}
SPL {X  -165.650, Y  +587.996, Z    +0.000, E1   -53.969, E3 +279139.421}
SPL {X  -165.650, Y  +595.185, Z    +0.000, E1   -53.962, E3 +279150.130}
SPL {X  -165.650, Y  +602.138, Z    +0.000, E1   -53.941, E3 +279160.625}
SPL {X  -165.650, Y  +610.307, Z    +0.000, E1   -53.995, E3 +279172.472}
SPL {X  -165.650, Y  +617.878, Z    +0.000, E1   -53.838, E3 +279184.729}
SPL {X  -165.650, Y  +626.374, Z    +0.000, E1   -54.092, E3 +279195.744}
SPL {X  -165.650, Y  +632.964, Z    +0.000, E1   -53.887, E3 +279206.872}
SPL {X  -165.650, Y  +640.262, Z    +0.000, E1   -53.965, E3 +279217.187}
SPL {X  -165.650, Y  +647.911, Z    +0.000, E1   -53.930, E3 +279228.941}
SPL {X  -165.650, Y  +656.836, Z    +0.000, E1   -54.184, E3 +279240.473}
SPL {X  -165.650, Y  +659.513, Z    +0.000, E1   -53.578, E3 +279248.203}
SPL {X  -165.650, Y  +667.820, Z    +0.000, E1   -53.975, E3 +279258.268}
SPL {X  -165.623, Y  +678.503, Z    +0.000, E1   -53.932, E3 +279274.619}
SPL {X  -165.027, Y  +689.850, Z    +0.000, E1   -53.862, E3 +279291.883}
SPL {X  -163.840, Y  +699.919, Z    +0.000, E1   -53.732, E3 +279307.665}
SPL {X  -162.702, Y  +706.614, Z    +0.000, E1   -53.230, E3 +279320.516}
SPL {X  -161.265, Y  +713.361, Z    +0.000, E1   -53.436, E3 +279329.325}
SPL {X  -159.936, Y  +718.632, Z    +0.000, E1   -52.857, E3 +279340.654}
SPL {X  -157.868, Y  +725.674, Z    +0.000, E1   -52.862, E3 +279350.995}
SPL {X  -156.314, Y  +730.327, Z    +0.000, E1   -52.199, E3 +279361.676}
SPL {X  -153.975, Y  +736.588, Z    +0.000, E1   -51.877, E3 +279372.707}
SPL {X  -151.949, Y  +741.465, Z    +0.000, E1   -51.645, E3 +279381.112}
SPL {X  -149.075, Y  +747.727, Z    +0.000, E1   -52.134, E3 +279387.827}
SPL {X  -137.775, Y  +767.467, Z    +0.000, E1   -56.912, E3 +279390.490}
SPL {X  -128.847, Y  +779.607, Z    +0.000, E1   -49.118, E3 +279465.506}
SPL {X   -94.133, Y  +811.804, Z    +0.000, E1   -53.019, E3 +279520.141}
ENDSPLINE

SPLINE
SPL {X  -134.098, Y  +772.750, Z    +0.000, E1   -45.587, E3 +279595.435}
SPL {X  -155.319, Y  +733.085, Z    +0.000, E1   -31.947, E3 +279586.313}
SPL {X  -162.077, Y  +709.719, Z    +0.000, E1   -21.590, E3 +279587.990}
SPL {X  -164.499, Y  +694.994, Z    +0.000, E1   -13.860, E3 +279588.775}
SPL {X  -165.513, Y  +682.236, Z    +0.000, E1    -6.385, E3 +279587.111}
SPL {X  -165.650, Y  +675.776, Z    +0.000, E1    -2.014, E3 +279586.418}
SPL {X  -165.650, Y  +672.938, Z    +0.000, E1    +0.157, E3 +279585.434}
SPL {X  -165.650, Y  +669.402, Z    +0.000, E1    +3.448, E3 +279584.825}
SPL {X  -165.650, Y  +663.061, Z    +0.000, E1   +11.076, E3 +279583.819}
SPL {X  -165.650, Y  +656.573, Z    +0.000, E1   +19.875, E3 +279583.626}
SPL {X  -165.650, Y  +650.769, Z    +0.000, E1   +28.083, E3 +279581.992}
SPL {X  -165.650, Y  +639.700, Z    +0.000, E1   +43.326, E3 +279577.054}
SPL {X  -165.650, Y  +605.320, Z    +0.000, E1   +76.562, E3 +279556.463}
SPL {X  -165.650, Y  +597.745, Z    +0.000, E1   +59.636, E3 +279594.464}
SPL {X  -165.650, Y  +596.360, Z    +0.000, E1   +54.978, E3 +279608.072}
SPL {X  -165.650, Y  +521.429, Z    +0.000, E1   +61.144, E3 +279661.303}
ENDSPLINE

SPLINE
SPL {X  -165.650, Y  +526.028, Z    +0.000, E1   +58.071, E3 +279675.078}
SPL {X  -165.650, Y  +539.856, Z    +0.000, E1   +53.398, E3 +279685.626}
ENDSPLINE

SPLINE
SPL {X  -165.650, Y  +532.042, Z    +0.000, E1   +53.611, E3 +279696.097}
SPL {X  -165.650, Y  +526.147, Z    +0.000, E1   +53.495, E3 +279705.736}
SPL {X  -165.650, Y  +517.365, Z    +0.000, E1   +53.387, E3 +279719.904}
SPL {X  -165.650, Y  +505.685, Z    +0.000, E1   +53.701, E3 +279735.529}
SPL {X  -165.650, Y  +498.275, Z    +0.000, E1   +53.357, E3 +279748.837}
SPL {X  -165.650, Y  +487.031, Z    +0.000, E1   +53.931, E3 +279762.246}
SPL {X  -165.650, Y  +450.615, Z    +0.000, E1   +59.721, E3 +279773.486}
SPL {X  -165.650, Y  +449.326, Z    +0.000, E1   +58.606, E3 +279782.535}
SPL {X  -165.650, Y  +442.154, Z    +0.000, E1   +58.369, E3 +279793.159}
SPL {X  -165.650, Y  +437.405, Z    +0.000, E1   +57.663, E3 +279803.769}
SPL {X  -165.650, Y  +432.227, Z    +0.000, E1   +57.103, E3 +279814.256}
SPL {X  -165.650, Y  +428.683, Z    +0.000, E1   +56.222, E3 +279824.611}
SPL {X  -165.650, Y  +424.202, Z    +0.000, E1   +55.382, E3 +279836.300}
SPL {X  -165.650, Y  +418.756, Z    +0.000, E1   +54.154, E3 +279851.979}
SPL {X  -165.650, Y  +410.508, Z    +0.000, E1   +54.007, E3 +279864.934}
SPL {X  -165.650, Y  +403.104, Z    +0.000, E1   +53.908, E3 +279876.716}
SPL {X  -165.650, Y  +393.046, Z    +0.000, E1   +53.951, E3 +279891.399}
SPL {X  -165.650, Y  +383.306, Z    +0.000, E1   +53.987, E3 +279905.676}
SPL {X  -165.640, Y  +376.676, Z    +0.000, E1   +53.760, E3 +279916.843}
SPL {X  -165.408, Y  +369.556, Z    +0.000, E1   +53.942, E3 +279926.394}
SPL {X  -164.927, Y  +363.041, Z    +0.000, E1   +53.687, E3 +279937.690}
SPL {X  -163.980, Y  +355.035, Z    +0.000, E1   +53.657, E3 +279949.886}
SPL {X  -162.665, Y  +347.197, Z    +0.000, E1   +53.396, E3 +279963.149}
SPL {X  -161.218, Y  +340.437, Z    +0.000, E1   +53.207, E3 +279974.248}
SPL {X  -159.523, Y  +333.864, Z    +0.000, E1   +52.908, E3 +279985.870}
SPL {X  -157.624, Y  +327.563, Z    +0.000, E1   +52.705, E3 +279996.280}
SPL {X  -156.289, Y  +323.602, Z    +0.000, E1   +52.159, E3 +280005.168}
SPL {X  -153.877, Y  +317.168, Z    +0.000, E1   +51.945, E3 +280016.030}
SPL {X  -151.035, Y  +310.467, Z    +0.000, E1   +51.312, E3 +280029.275}
SPL {X  -139.567, Y  +289.276, Z    +0.000, E1   +56.334, E3 +280033.363}
SPL {X  -117.053, Y  +261.289, Z    +0.000, E1   +49.815, E3 +280146.897}
ENDSPLINE

SPLINE
SPL {X  -148.836, Y  +305.783, Z    +0.000, E1   +38.029, E3 +280238.375}
SPL {X  -161.816, Y  +343.065, Z    +0.000, E1   +22.147, E3 +280229.025}
SPL {X  -164.614, Y  +360.007, Z    +0.000, E1   +13.213, E3 +280224.811}
SPL {X  -165.520, Y  +371.933, Z    +0.000, E1    +6.276, E3 +280227.565}
SPL {X  -165.650, Y  +378.704, Z    +0.000, E1    +1.700, E3 +280226.435}
SPL {X  -165.650, Y  +382.197, Z    +0.000, E1    -1.038, E3 +280225.508}
SPL {X  -165.650, Y  +386.782, Z    +0.000, E1    -5.783, E3 +280224.986}
SPL {X  -165.650, Y  +392.406, Z    +0.000, E1   -13.042, E3 +280222.883}
SPL {X  -165.650, Y  +400.489, Z    +0.000, E1   -23.243, E3 +280224.047}
SPL {X  -165.650, Y  +415.469, Z    +0.000, E1   -43.461, E3 +280218.455}
SPL {X  -165.650, Y  +460.095, Z    +0.000, E1   -60.221, E3 +280236.717}
SPL {X  -165.650, Y  +535.749, Z    +0.000, E1   -60.559, E3 +280307.560}
ENDSPLINE

SPLINE
SPL {X  -165.650, Y  +516.866, Z    +0.000, E1   -54.768, E3 +280320.110}
ENDSPLINE

SPLINE
SPL {X  -165.650, Y  +521.328, Z    +0.000, E1   -53.870, E3 +280332.402}
SPL {X  -165.650, Y  +531.171, Z    +0.000, E1   -54.075, E3 +280345.746}
SPL {X  -165.650, Y  +538.771, Z    +0.000, E1   -53.840, E3 +280358.486}
SPL {X  -165.650, Y  +548.103, Z    +0.000, E1   -53.944, E3 +280371.833}
SPL {X  -165.650, Y  +558.071, Z    +0.000, E1   -53.870, E3 +280387.174}
SPL {X  -165.650, Y  +568.053, Z    +0.000, E1   -54.124, E3 +280400.351}
SPL {X  -165.650, Y  +577.021, Z    +0.000, E1   -53.813, E3 +280415.850}
SPL {X  -165.650, Y  +587.996, Z    +0.000, E1   -53.969, E3 +280431.088}
SPL {X  -165.650, Y  +595.185, Z    +0.000, E1   -53.962, E3 +280441.797}
SPL {X  -165.650, Y  +602.138, Z    +0.000, E1   -53.941, E3 +280452.291}
SPL {X  -165.650, Y  +610.307, Z    +0.000, E1   -53.995, E3 +280464.139}
SPL {X  -165.650, Y  +617.878, Z    +0.000, E1   -53.838, E3 +280476.396}
SPL {X  -165.650, Y  +627.853, Z    +0.000, E1   -53.937, E3 +280490.749}
SPL {X  -165.650, Y  +638.510, Z    +0.000, E1   -54.057, E3 +280505.809}
SPL {X  -165.650, Y  +647.911, Z    +0.000, E1   -53.930, E3 +280520.608}
SPL {X  -165.650, Y  +658.189, Z    +0.000, E1   -53.932, E3 +280535.908}
SPL {X  -165.650, Y  +667.820, Z    +0.000, E1   -53.975, E3 +280549.934}
SPL {X  -165.623, Y  +678.503, Z    +0.000, E1   -53.932, E3 +280566.286}
SPL {X  -165.171, Y  +688.090, Z    +0.000, E1   -54.025, E3 +280579.734}
SPL {X  -164.558, Y  +694.489, Z    +0.000, E1   -53.745, E3 +280591.083}
SPL {X  -163.580, Y  +701.606, Z    +0.000, E1   -53.591, E3 +280602.516}
SPL {X  -162.702, Y  +706.614, Z    +0.000, E1   -53.230, E3 +280612.183}
SPL {X  -160.941, Y  +714.715, Z    +0.000, E1   -53.321, E3 +280623.802}
SPL {X  -159.638, Y  +719.723, Z    +0.000, E1   -52.685, E3 +280634.805}
SPL {X  -157.521, Y  +726.754, Z    +0.000, E1   -52.585, E3 +280646.000}
SPL {X  -155.632, Y  +732.234, Z    +0.000, E1   -52.209, E3 +280656.047}
SPL {X  -153.975, Y  +736.588, Z    +0.000, E1   -51.877, E3 +280664.373}
SPL {X  -151.949, Y  +741.465, Z    +0.000, E1   -51.645, E3 +280672.779}
SPL {X  -149.075, Y  +747.727, Z    +0.000, E1   -52.134, E3 +280679.493}
SPL {X  -137.775, Y  +767.467, Z    +0.000, E1   -56.912, E3 +280682.157}
SPL {X  -128.847, Y  +779.607, Z    +0.000, E1   -49.118, E3 +280757.173}
SPL {X   -94.133, Y  +811.804, Z    +0.000, E1   -53.019, E3 +280811.807}
ENDSPLINE

SPLINE
SPL {X  -134.098, Y  +772.750, Z    +0.000, E1   -45.587, E3 +280887.102}
SPL {X  -155.319, Y  +733.085, Z    +0.000, E1   -31.947, E3 +280877.979}
SPL {X  -162.077, Y  +709.719, Z    +0.000, E1   -21.590, E3 +280879.657}
SPL {X  -164.499, Y  +694.994, Z    +0.000, E1   -13.860, E3 +280880.442}
SPL {X  -165.382, Y  +684.927, Z    +0.000, E1    -7.984, E3 +280878.619}
SPL {X  -165.645, Y  +676.778, Z    +0.000, E1    -2.777, E3 +280878.341}
SPL {X  -165.650, Y  +672.041, Z    +0.000, E1    +0.844, E3 +280877.033}
SPL {X  -165.650, Y  +667.328, Z    +0.000, E1    +5.806, E3 +280876.410}
SPL {X  -165.650, Y  +661.774, Z    +0.000, E1   +13.006, E3 +280874.734}
SPL {X  -165.650, Y  +656.573, Z    +0.000, E1   +19.875, E3 +280875.292}
SPL {X  -165.650, Y  +650.769, Z    +0.000, E1   +28.083, E3 +280873.658}
SPL {X  -165.650, Y  +639.700, Z    +0.000, E1   +43.326, E3 +280868.720}
SPL {X  -165.650, Y  +605.320, Z    +0.000, E1   +76.562, E3 +280848.130}
SPL {X  -165.650, Y  +597.745, Z    +0.000, E1   +59.636, E3 +280886.131}
SPL {X  -165.650, Y  +596.360, Z    +0.000, E1   +54.978, E3 +280899.739}
SPL {X  -165.650, Y  +521.429, Z    +0.000, E1   +61.144, E3 +280952.970}
ENDSPLINE

SPLINE
SPL {X  -165.650, Y  +526.028, Z    +0.000, E1   +58.071, E3 +280966.745}
SPL {X  -165.650, Y  +539.856, Z    +0.000, E1   +53.398, E3 +280977.292}
ENDSPLINE

SPLINE
SPL {X  -165.650, Y  +530.389, Z    +0.000, E1   +53.621, E3 +280990.298}
SPL {X  -165.650, Y  +521.849, Z    +0.000, E1   +53.452, E3 +281004.237}
SPL {X  -165.650, Y  +512.447, Z    +0.000, E1   +53.456, E3 +281018.497}
SPL {X  -165.650, Y  +503.994, Z    +0.000, E1   +53.652, E3 +281029.936}
SPL {X  -165.650, Y  +498.275, Z    +0.000, E1   +53.357, E3 +281040.504}
SPL {X  -165.650, Y  +491.031, Z    +0.000, E1   +53.348, E3 +281051.524}
SPL {X  -165.650, Y  +479.077, Z    +0.000, E1   +55.039, E3 +281058.647}
SPL {X  -165.650, Y  +450.615, Z    +0.000, E1   +59.721, E3 +281065.152}
SPL {X  -165.650, Y  +449.326, Z    +0.000, E1   +58.606, E3 +281074.202}
SPL {X  -165.650, Y  +442.154, Z    +0.000, E1   +58.369, E3 +281084.826}
SPL {X  -165.650, Y  +437.405, Z    +0.000, E1   +57.663, E3 +281095.435}
SPL {X  -165.650, Y  +432.227, Z    +0.000, E1   +57.103, E3 +281105.923}
SPL {X  -165.650, Y  +428.683, Z    +0.000, E1   +56.222, E3 +281116.277}
SPL {X  -165.650, Y  +424.202, Z    +0.000, E1   +55.382, E3 +281127.966}
SPL {X  -165.650, Y  +418.756, Z    +0.000, E1   +54.154, E3 +281143.645}
SPL {X  -165.650, Y  +410.508, Z    +0.000, E1   +54.007, E3 +281156.601}
SPL {X  -165.650, Y  +403.104, Z    +0.000, E1   +53.908, E3 +281168.382}
SPL {X  -165.650, Y  +393.046, Z    +0.000, E1   +53.951, E3 +281183.066}
SPL {X  -165.650, Y  +383.306, Z    +0.000, E1   +53.987, E3 +281197.343}
SPL {X  -165.640, Y  +376.676, Z    +0.000, E1   +53.760, E3 +281208.510}
SPL {X  -165.408, Y  +369.556, Z    +0.000, E1   +53.942, E3 +281218.061}
SPL {X  -164.927, Y  +363.041, Z    +0.000, E1   +53.687, E3 +281229.356}
SPL {X  -163.980, Y  +355.035, Z    +0.000, E1   +53.657, E3 +281241.553}
SPL {X  -162.665, Y  +347.197, Z    +0.000, E1   +53.396, E3 +281254.816}
SPL {X  -161.218, Y  +340.437, Z    +0.000, E1   +53.207, E3 +281265.915}
SPL {X  -159.523, Y  +333.864, Z    +0.000, E1   +52.908, E3 +281277.537}
SPL {X  -157.624, Y  +327.563, Z    +0.000, E1   +52.705, E3 +281287.946}
SPL {X  -156.289, Y  +323.602, Z    +0.000, E1   +52.159, E3 +281296.835}
SPL {X  -153.877, Y  +317.168, Z    +0.000, E1   +51.945, E3 +281307.696}
SPL {X  -151.035, Y  +310.467, Z    +0.000, E1   +51.312, E3 +281320.942}
SPL {X  -139.567, Y  +289.276, Z    +0.000, E1   +56.334, E3 +281325.030}
SPL {X  -117.053, Y  +261.289, Z    +0.000, E1   +49.815, E3 +281438.564}
ENDSPLINE

SPLINE
SPL {X  -148.836, Y  +305.783, Z    +0.000, E1   +38.029, E3 +281530.041}
SPL {X  -161.816, Y  +343.065, Z    +0.000, E1   +22.147, E3 +281520.691}
SPL {X  -164.614, Y  +360.007, Z    +0.000, E1   +13.213, E3 +281516.478}
SPL {X  -165.520, Y  +371.933, Z    +0.000, E1    +6.276, E3 +281519.232}
SPL {X  -165.650, Y  +380.164, Z    +0.000, E1    +0.707, E3 +281517.701}
SPL {X  -165.650, Y  +384.850, Z    +0.000, E1    -3.598, E3 +281516.809}
SPL {X  -165.650, Y  +391.255, Z    +0.000, E1   -11.346, E3 +281515.150}
SPL {X  -165.650, Y  +398.038, Z    +0.000, E1   -20.113, E3 +281516.117}
SPL {X  -165.650, Y  +403.005, Z    +0.000, E1   -26.762, E3 +281515.299}
SPL {X  -165.650, Y  +415.469, Z    +0.000, E1   -43.461, E3 +281510.122}
SPL {X  -165.650, Y  +460.095, Z    +0.000, E1   -60.221, E3 +281528.383}
SPL {X  -165.650, Y  +535.749, Z    +0.000, E1   -60.559, E3 +281599.227}
ENDSPLINE

SPLINE
SPL {X  -165.650, Y  +516.750, Z    +0.000, E1   -54.244, E3 +281615.077}
ENDSPLINE

SPLINE
SPL {X  -165.650, Y  +524.345, Z    +0.000, E1   -54.115, E3 +281626.974}
SPL {X  -165.650, Y  +531.171, Z    +0.000, E1   -54.075, E3 +281637.413}
SPL {X  -165.650, Y  +538.771, Z    +0.000, E1   -53.840, E3 +281650.153}
SPL {X  -165.650, Y  +545.884, Z    +0.000, E1   -53.883, E3 +281660.458}
SPL {X  -165.650, Y  +553.081, Z    +0.000, E1   -53.834, E3 +281671.591}
SPL {X  -165.650, Y  +560.989, Z    +0.000, E1   -53.974, E3 +281682.428}
SPL {X  -165.650, Y  +568.053, Z    +0.000, E1   -54.124, E3 +281692.018}
SPL {X  -165.650, Y  +577.021, Z    +0.000, E1   -53.813, E3 +281707.517}
SPL {X  -165.650, Y  +587.996, Z    +0.000, E1   -53.969, E3 +281722.754}
SPL {X  -165.650, Y  +595.185, Z    +0.000, E1   -53.962, E3 +281733.464}
SPL {X  -165.650, Y  +602.138, Z    +0.000, E1   -53.941, E3 +281743.958}
SPL {X  -165.650, Y  +610.307, Z    +0.000, E1   -53.995, E3 +281755.806}
SPL {X  -165.650, Y  +617.878, Z    +0.000, E1   -53.838, E3 +281768.062}
SPL {X  -165.650, Y  +627.853, Z    +0.000, E1   -53.937, E3 +281782.416}
SPL {X  -165.650, Y  +638.510, Z    +0.000, E1   -54.057, E3 +281797.476}
SPL {X  -165.650, Y  +645.417, Z    +0.000, E1   -53.856, E3 +281808.889}
SPL {X  -165.650, Y  +654.069, Z    +0.000, E1   -54.108, E3 +281820.309}
SPL {X  -165.650, Y  +659.513, Z    +0.000, E1   -53.578, E3 +281831.536}
SPL {X  -165.650, Y  +667.820, Z    +0.000, E1   -53.975, E3 +281841.601}
SPL {X  -165.650, Y  +674.957, Z    +0.000, E1   -53.977, E3 +281852.113}
SPL {X  -165.574, Y  +680.515, Z    +0.000, E1   -53.820, E3 +281861.440}
SPL {X  -165.171, Y  +688.090, Z    +0.000, E1   -54.025, E3 +281871.400}
SPL {X  -164.558, Y  +694.489, Z    +0.000, E1   -53.745, E3 +281882.750}
SPL {X  -163.580, Y  +701.606, Z    +0.000, E1   -53.591, E3 +281894.183}
SPL {X  -162.702, Y  +706.614, Z    +0.000, E1   -53.230, E3 +281903.849}
SPL {X  -160.941, Y  +714.715, Z    +0.000, E1   -53.321, E3 +281915.469}
SPL {X  -159.638, Y  +719.723, Z    +0.000, E1   -52.685, E3 +281926.471}
SPL {X  -157.521, Y  +726.754, Z    +0.000, E1   -52.585, E3 +281937.667}
SPL {X  -155.632, Y  +732.234, Z    +0.000, E1   -52.209, E3 +281947.714}
SPL {X  -153.975, Y  +736.588, Z    +0.000, E1   -51.877, E3 +281956.040}
SPL {X  -151.949, Y  +741.465, Z    +0.000, E1   -51.645, E3 +281964.445}
SPL {X  -149.075, Y  +747.727, Z    +0.000, E1   -52.134, E3 +281971.160}
SPL {X  -137.775, Y  +767.467, Z    +0.000, E1   -56.912, E3 +281973.823}
SPL {X  -128.847, Y  +779.607, Z    +0.000, E1   -49.118, E3 +282048.840}
SPL {X   -94.133, Y  +811.804, Z    +0.000, E1   -53.019, E3 +282103.474}
ENDSPLINE

SPLINE
SPL {X  -134.098, Y  +772.750, Z    +0.000, E1   -45.587, E3 +282178.768}
SPL {X  -155.319, Y  +733.085, Z    +0.000, E1   -31.947, E3 +282169.646}
SPL {X  -162.077, Y  +709.719, Z    +0.000, E1   -21.590, E3 +282171.324}
SPL {X  -164.499, Y  +694.994, Z    +0.000, E1   -13.860, E3 +282172.108}
SPL {X  -165.513, Y  +682.236, Z    +0.000, E1    -6.385, E3 +282170.444}
SPL {X  -165.650, Y  +675.776, Z    +0.000, E1    -2.014, E3 +282169.752}
SPL {X  -165.650, Y  +672.041, Z    +0.000, E1    +0.844, E3 +282168.700}
SPL {X  -165.650, Y  +667.328, Z    +0.000, E1    +5.806, E3 +282168.076}
SPL {X  -165.650, Y  +661.774, Z    +0.000, E1   +13.006, E3 +282166.400}
SPL {X  -165.650, Y  +654.085, Z    +0.000, E1   +23.232, E3 +282166.260}
SPL {X  -165.650, Y  +639.700, Z    +0.000, E1   +43.326, E3 +282160.387}
SPL {X  -165.650, Y  +605.320, Z    +0.000, E1   +76.562, E3 +282139.796}
SPL {X  -165.650, Y  +596.505, Z    +0.000, E1   +55.802, E3 +282189.152}
SPL {X  -165.650, Y  +524.050, Z    +0.000, E1   +59.300, E3 +282253.312}
ENDSPLINE

SPLINE
SPL {X  -165.650, Y  +539.856, Z    +0.000, E1   +53.398, E3 +282268.959}
ENDSPLINE

SPLINE
SPL {X  -165.650, Y  +530.389, Z    +0.000, E1   +53.621, E3 +282281.964}
SPL {X  -165.650, Y  +521.849, Z    +0.000, E1   +53.452, E3 +282295.904}
SPL {X  -165.650, Y  +515.134, Z    +0.000, E1   +53.252, E3 +282307.255}
SPL {X  -165.650, Y  +505.685, Z    +0.000, E1   +53.701, E3 +282318.863}
SPL {X  -165.650, Y  +498.275, Z    +0.000, E1   +53.357, E3 +282332.170}
SPL {X  -165.650, Y  +487.031, Z    +0.000, E1   +53.931, E3 +282345.579}
SPL {X  -165.650, Y  +450.615, Z    +0.000, E1   +59.721, E3 +282356.819}
SPL {X  -165.650, Y  +449.326, Z    +0.000, E1   +58.606, E3 +282365.868}
SPL {X  -165.650, Y  +442.154, Z    +0.000, E1   +58.369, E3 +282376.492}
SPL {X  -165.650, Y  +437.405, Z    +0.000, E1   +57.663, E3 +282387.102}
SPL {X  -165.650, Y  +432.227, Z    +0.000, E1   +57.103, E3 +282397.590}
SPL {X  -165.650, Y  +428.683, Z    +0.000, E1   +56.222, E3 +282407.944}
SPL {X  -165.650, Y  +424.202, Z    +0.000, E1   +55.382, E3 +282419.633}
SPL {X  -165.650, Y  +418.469, Z    +0.000, E1   +54.594, E3 +282432.741}
SPL {X  -165.650, Y  +413.857, Z    +0.000, E1   +53.683, E3 +282445.312}
SPL {X  -165.650, Y  +405.379, Z    +0.000, E1   +53.922, E3 +282456.426}
SPL {X  -165.650, Y  +400.791, Z    +0.000, E1   +53.827, E3 +282463.840}
SPL {X  -165.650, Y  +391.401, Z    +0.000, E1   +53.934, E3 +282477.440}
SPL {X  -165.650, Y  +378.987, Z    +0.000, E1   +53.974, E3 +282495.636}
SPL {X  -165.408, Y  +369.556, Z    +0.000, E1   +53.942, E3 +282509.727}
SPL {X  -164.927, Y  +363.041, Z    +0.000, E1   +53.687, E3 +282521.023}
SPL {X  -164.096, Y  +355.862, Z    +0.000, E1   +53.838, E3 +282530.753}
SPL {X  -163.142, Y  +349.785, Z    +0.000, E1   +53.493, E3 +282541.969}
SPL {X  -161.604, Y  +342.113, Z    +0.000, E1   +53.155, E3 +282555.463}
SPL {X  -159.523, Y  +333.864, Z    +0.000, E1   +52.908, E3 +282569.204}
SPL {X  -157.624, Y  +327.563, Z    +0.000, E1   +52.705, E3 +282579.613}
SPL {X  -155.665, Y  +321.859, Z    +0.000, E1   +52.064, E3 +282591.786}
SPL {X  -152.682, Y  +314.249, Z    +0.000, E1   +51.841, E3 +282604.234}
SPL {X  -150.607, Y  +309.525, Z    +0.000, E1   +51.147, E3 +282614.719}
SPL {X  -139.567, Y  +289.276, Z    +0.000, E1   +56.334, E3 +282616.697}
SPL {X  -116.936, Y  +261.172, Z    +0.000, E1   +51.023, E3 +282706.813}
ENDSPLINE

SPLINE
SPL {X  -117.298, Y  +261.533, Z    +0.000, E1   +49.535, E3 +282735.589}
SPL {X  -148.836, Y  +305.783, Z    +0.000, E1   +38.029, E3 +282821.708}
SPL {X  -161.816, Y  +343.065, Z    +0.000, E1   +22.147, E3 +282812.358}
SPL {X  -164.614, Y  +360.007, Z    +0.000, E1   +13.213, E3 +282808.144}
SPL {X  -165.520, Y  +371.933, Z    +0.000, E1    +6.276, E3 +282810.899}
SPL {X  -165.650, Y  +380.164, Z    +0.000, E1    +0.707, E3 +282809.368}
SPL {X  -165.650, Y  +383.228, Z    +0.000, E1    -2.108, E3 +282808.593}
SPL {X  -165.650, Y  +386.782, Z    +0.000, E1    -5.783, E3 +282808.319}
SPL {X  -165.650, Y  +392.406, Z    +0.000, E1   -13.042, E3 +282806.216}
SPL {X  -165.650, Y  +400.489, Z    +0.000, E1   -23.243, E3 +282807.380}
SPL {X  -165.650, Y  +415.469, Z    +0.000, E1   -43.461, E3 +282801.789}
SPL {X  -165.650, Y  +452.083, Z    +0.000, E1   -59.895, E3 +282813.702}
SPL {X  -165.650, Y  +462.893, Z    +0.000, E1   -60.288, E3 +282822.284}
SPL {X  -165.650, Y  +535.749, Z    +0.000, E1   -60.559, E3 +282890.894}
ENDSPLINE

SPLINE
SPL {X  -165.650, Y  +516.750, Z    +0.000, E1   -54.244, E3 +282906.744}
ENDSPLINE

SPLINE
SPL {X  -165.650, Y  +524.345, Z    +0.000, E1   -54.115, E3 +282918.641}
SPL {X  -165.650, Y  +531.171, Z    +0.000, E1   -54.075, E3 +282929.079}
SPL {X  -165.650, Y  +538.771, Z    +0.000, E1   -53.840, E3 +282941.820}
SPL {X  -165.650, Y  +548.103, Z    +0.000, E1   -53.944, E3 +282955.166}
SPL {X  -165.650, Y  +558.071, Z    +0.000, E1   -53.870, E3 +282970.507}
SPL {X  -165.650, Y  +568.053, Z    +0.000, E1   -54.124, E3 +282983.685}
SPL {X  -165.650, Y  +577.021, Z    +0.000, E1   -53.813, E3 +282999.183}
SPL {X  -165.650, Y  +587.996, Z    +0.000, E1   -53.969, E3 +283014.421}
SPL {X  -165.650, Y  +595.185, Z    +0.000, E1   -53.962, E3 +283025.130}
SPL {X  -165.650, Y  +602.138, Z    +0.000, E1   -53.941, E3 +283035.625}
SPL {X  -165.650, Y  +610.307, Z    +0.000, E1   -53.995, E3 +283047.472}
SPL {X  -165.650, Y  +617.878, Z    +0.000, E1   -53.838, E3 +283059.729}
SPL {X  -165.650, Y  +627.853, Z    +0.000, E1   -53.937, E3 +283074.083}
SPL {X  -165.650, Y  +638.510, Z    +0.000, E1   -54.057, E3 +283089.142}
SPL {X  -165.650, Y  +647.911, Z    +0.000, E1   -53.930, E3 +283103.941}
SPL {X  -165.650, Y  +656.836, Z    +0.000, E1   -54.184, E3 +283115.473}
SPL {X  -165.650, Y  +659.513, Z    +0.000, E1   -53.578, E3 +283123.203}
SPL {X  -165.650, Y  +667.820, Z    +0.000, E1   -53.975, E3 +283133.268}
SPL {X  -165.650, Y  +674.957, Z    +0.000, E1   -53.977, E3 +283143.780}
SPL {X  -165.574, Y  +680.515, Z    +0.000, E1   -53.820, E3 +283153.107}
SPL {X  -165.027, Y  +689.850, Z    +0.000, E1   -53.862, E3 +283166.883}
SPL {X  -163.840, Y  +699.919, Z    +0.000, E1   -53.732, E3 +283182.665}
SPL {X  -162.702, Y  +706.614, Z    +0.000, E1   -53.230, E3 +283195.516}
SPL {X  -160.941, Y  +714.715, Z    +0.000, E1   -53.321, E3 +283207.136}
SPL {X  -159.638, Y  +719.723, Z    +0.000, E1   -52.685, E3 +283218.138}
SPL {X  -157.868, Y  +725.674, Z    +0.000, E1   -52.862, E3 +283225.995}
SPL {X  -156.314, Y  +730.327, Z    +0.000, E1   -52.199, E3 +283236.676}
SPL {X  -153.975, Y  +736.588, Z    +0.000, E1   -51.877, E3 +283247.707}
SPL {X  -151.181, Y  +743.207, Z    +0.000, E1   -51.549, E3 +283259.327}
SPL {X  -146.528, Y  +752.763, Z    +0.000, E1   -53.481, E3 +283263.505}
SPL {X  -137.775, Y  +767.467, Z    +0.000, E1   -56.912, E3 +283265.490}
SPL {X  -128.847, Y  +779.607, Z    +0.000, E1   -49.118, E3 +283340.506}
SPL {X   -94.133, Y  +811.804, Z    +0.000, E1   -53.019, E3 +283395.141}
ENDSPLINE

SPLINE
SPL {X  -134.098, Y  +772.750, Z    +0.000, E1   -45.587, E3 +283470.435}
SPL {X  -155.319, Y  +733.085, Z    +0.000, E1   -31.947, E3 +283461.313}
SPL {X  -162.077, Y  +709.719, Z    +0.000, E1   -21.590, E3 +283462.990}
SPL {X  -164.499, Y  +694.994, Z    +0.000, E1   -13.860, E3 +283463.775}
SPL {X  -165.382, Y  +684.927, Z    +0.000, E1    -7.984, E3 +283461.952}
SPL {X  -165.645, Y  +676.778, Z    +0.000, E1    -2.777, E3 +283461.675}
SPL {X  -165.650, Y  +672.938, Z    +0.000, E1    +0.157, E3 +283460.434}
SPL {X  -165.650, Y  +670.852, Z    +0.000, E1    +2.095, E3 +283460.277}
SPL {X  -165.650, Y  +667.328, Z    +0.000, E1    +5.806, E3 +283459.743}
SPL {X  -165.650, Y  +661.774, Z    +0.000, E1   +13.006, E3 +283458.067}
SPL {X  -165.650, Y  +656.573, Z    +0.000, E1   +19.875, E3 +283458.626}
SPL {X  -165.650, Y  +650.769, Z    +0.000, E1   +28.083, E3 +283456.992}
SPL {X  -165.650, Y  +639.700, Z    +0.000, E1   +43.326, E3 +283452.054}
SPL {X  -165.650, Y  +605.320, Z    +0.000, E1   +76.562, E3 +283431.463}
SPL {X  -165.650, Y  +597.745, Z    +0.000, E1   +59.636, E3 +283469.464}
SPL {X  -165.650, Y  +596.360, Z    +0.000, E1   +54.978, E3 +283483.072}
SPL {X  -165.650, Y  +521.429, Z    +0.000, E1   +61.144, E3 +283536.303}
ENDSPLINE

SPLINE
SPL {X  -165.650, Y  +526.028, Z    +0.000, E1   +58.071, E3 +283550.078}
SPL {X  -165.650, Y  +539.856, Z    +0.000, E1   +53.398, E3 +283560.626}
ENDSPLINE

SPLINE
SPL {X  -165.650, Y  +532.042, Z    +0.000, E1   +53.611, E3 +283571.097}
SPL {X  -165.650, Y  +526.147, Z    +0.000, E1   +53.495, E3 +283580.736}
SPL {X  -165.650, Y  +517.365, Z    +0.000, E1   +53.387, E3 +283594.904}
SPL {X  -165.650, Y  +505.685, Z    +0.000, E1   +53.701, E3 +283610.529}
SPL {X  -165.650, Y  +498.275, Z    +0.000, E1   +53.357, E3 +283623.837}
SPL {X  -165.650, Y  +487.031, Z    +0.000, E1   +53.931, E3 +283637.246}
SPL {X  -165.650, Y  +450.615, Z    +0.000, E1   +59.721, E3 +283648.486}
SPL {X  -165.650, Y  +449.326, Z    +0.000, E1   +58.606, E3 +283657.535}
SPL {X  -165.650, Y  +442.154, Z    +0.000, E1   +58.369, E3 +283668.159}
SPL {X  -165.650, Y  +437.405, Z    +0.000, E1   +57.663, E3 +283678.769}
SPL {X  -165.650, Y  +432.227, Z    +0.000, E1   +57.103, E3 +283689.256}
SPL {X  -165.650, Y  +428.683, Z    +0.000, E1   +56.222, E3 +283699.611}
SPL {X  -165.650, Y  +424.202, Z    +0.000, E1   +55.382, E3 +283711.300}
SPL {X  -165.650, Y  +418.469, Z    +0.000, E1   +54.594, E3 +283724.408}
SPL {X  -165.650, Y  +413.857, Z    +0.000, E1   +53.683, E3 +283736.979}
SPL {X  -165.650, Y  +403.104, Z    +0.000, E1   +53.908, E3 +283751.716}
SPL {X  -165.650, Y  +391.401, Z    +0.000, E1   +53.934, E3 +283769.106}
SPL {X  -165.650, Y  +378.987, Z    +0.000, E1   +53.974, E3 +283787.303}
SPL {X  -165.408, Y  +369.556, Z    +0.000, E1   +53.942, E3 +283801.394}
SPL {X  -164.927, Y  +363.041, Z    +0.000, E1   +53.687, E3 +283812.690}
SPL {X  -164.096, Y  +355.862, Z    +0.000, E1   +53.838, E3 +283822.420}
SPL {X  -163.142, Y  +349.785, Z    +0.000, E1   +53.493, E3 +283833.636}
SPL {X  -161.604, Y  +342.113, Z    +0.000, E1   +53.155, E3 +283847.130}
SPL {X  -159.523, Y  +333.864, Z    +0.000, E1   +52.908, E3 +283860.870}
SPL {X  -157.624, Y  +327.563, Z    +0.000, E1   +52.705, E3 +283871.280}
SPL {X  -156.289, Y  +323.602, Z    +0.000, E1   +52.159, E3 +283880.168}
SPL {X  -154.898, Y  +319.792, Z    +0.000, E1   +51.850, E3 +283887.504}
SPL {X  -152.682, Y  +314.249, Z    +0.000, E1   +51.841, E3 +283895.901}
SPL {X  -150.607, Y  +309.525, Z    +0.000, E1   +51.147, E3 +283906.385}
SPL {X  -139.567, Y  +289.276, Z    +0.000, E1   +56.334, E3 +283908.363}
SPL {X  -117.053, Y  +261.289, Z    +0.000, E1   +49.815, E3 +284021.897}
ENDSPLINE

SPLINE
SPL {X  -148.836, Y  +305.783, Z    +0.000, E1   +38.029, E3 +284113.375}
SPL {X  -161.816, Y  +343.065, Z    +0.000, E1   +22.147, E3 +284104.025}
SPL {X  -164.614, Y  +360.007, Z    +0.000, E1   +13.213, E3 +284099.811}
SPL {X  -165.520, Y  +371.933, Z    +0.000, E1    +6.276, E3 +284102.565}
SPL {X  -165.650, Y  +380.164, Z    +0.000, E1    +0.707, E3 +284101.035}
SPL {X  -165.650, Y  +384.850, Z    +0.000, E1    -3.598, E3 +284100.142}
SPL {X  -165.650, Y  +391.255, Z    +0.000, E1   -11.346, E3 +284098.484}
SPL {X  -165.650, Y  +398.038, Z    +0.000, E1   -20.113, E3 +284099.450}
SPL {X  -165.650, Y  +403.005, Z    +0.000, E1   -26.762, E3 +284098.632}
SPL {X  -165.650, Y  +415.469, Z    +0.000, E1   -43.461, E3 +284093.455}
SPL {X  -165.650, Y  +460.095, Z    +0.000, E1   -60.221, E3 +284111.717}
SPL {X  -165.650, Y  +535.749, Z    +0.000, E1   -60.559, E3 +284182.560}
ENDSPLINE

SPLINE
SPL {X  -165.650, Y  +516.866, Z    +0.000, E1   -54.768, E3 +284195.110}
ENDSPLINE

SPLINE
SPL {X  -165.650, Y  +521.328, Z    +0.000, E1   -53.870, E3 +284207.402}
SPL {X  -165.650, Y  +531.171, Z    +0.000, E1   -54.075, E3 +284220.746}
SPL {X  -165.650, Y  +538.771, Z    +0.000, E1   -53.840, E3 +284233.486}
SPL {X  -165.650, Y  +545.884, Z    +0.000, E1   -53.883, E3 +284243.791}
SPL {X  -165.650, Y  +553.081, Z    +0.000, E1   -53.834, E3 +284254.924}
SPL {X  -165.650, Y  +560.989, Z    +0.000, E1   -53.974, E3 +284265.761}
SPL {X  -165.650, Y  +568.053, Z    +0.000, E1   -54.124, E3 +284275.351}
SPL {X  -165.650, Y  +577.021, Z    +0.000, E1   -53.813, E3 +284290.850}
SPL {X  -165.650, Y  +587.996, Z    +0.000, E1   -53.969, E3 +284306.088}
SPL {X  -165.650, Y  +595.185, Z    +0.000, E1   -53.962, E3 +284316.797}
SPL {X  -165.650, Y  +602.138, Z    +0.000, E1   -53.941, E3 +284327.291}
SPL {X  -165.650, Y  +610.307, Z    +0.000, E1   -53.995, E3 +284339.139}
SPL {X  -165.650, Y  +617.878, Z    +0.000, E1   -53.838, E3 +284351.396}
SPL {X  -165.650, Y  +627.853, Z    +0.000, E1   -53.937, E3 +284365.749}
SPL {X  -165.650, Y  +638.510, Z    +0.000, E1   -54.057, E3 +284380.809}
SPL {X  -165.650, Y  +647.911, Z    +0.000, E1   -53.930, E3 +284395.608}
SPL {X  -165.650, Y  +656.836, Z    +0.000, E1   -54.184, E3 +284407.140}
SPL {X  -165.650, Y  +659.513, Z    +0.000, E1   -53.578, E3 +284414.869}
SPL {X  -165.650, Y  +667.820, Z    +0.000, E1   -53.975, E3 +284424.934}
SPL {X  -165.623, Y  +678.503, Z    +0.000, E1   -53.932, E3 +284441.286}
SPL {X  -165.171, Y  +688.090, Z    +0.000, E1   -54.025, E3 +284454.734}
SPL {X  -164.558, Y  +694.489, Z    +0.000, E1   -53.745, E3 +284466.083}
SPL {X  -163.580, Y  +701.606, Z    +0.000, E1   -53.591, E3 +284477.516}
SPL {X  -162.702, Y  +706.614, Z    +0.000, E1   -53.230, E3 +284487.183}
SPL {X  -160.941, Y  +714.715, Z    +0.000, E1   -53.321, E3 +284498.802}
SPL {X  -159.638, Y  +719.723, Z    +0.000, E1   -52.685, E3 +284509.805}
SPL {X  -157.521, Y  +726.754, Z    +0.000, E1   -52.585, E3 +284521.000}
SPL {X  -155.632, Y  +732.234, Z    +0.000, E1   -52.209, E3 +284531.047}
SPL {X  -153.975, Y  +736.588, Z    +0.000, E1   -51.877, E3 +284539.373}
SPL {X  -151.949, Y  +741.465, Z    +0.000, E1   -51.645, E3 +284547.779}
SPL {X  -149.075, Y  +747.727, Z    +0.000, E1   -52.134, E3 +284554.493}
SPL {X  -137.775, Y  +767.467, Z    +0.000, E1   -56.912, E3 +284557.157}
SPL {X  -128.847, Y  +779.607, Z    +0.000, E1   -49.118, E3 +284632.173}
SPL {X   -94.133, Y  +811.804, Z    +0.000, E1   -53.019, E3 +284686.807}
ENDSPLINE

SPLINE
SPL {X  -134.098, Y  +772.750, Z    +0.000, E1   -45.587, E3 +284762.102}
SPL {X  -155.319, Y  +733.085, Z    +0.000, E1   -31.947, E3 +284752.979}
SPL {X  -162.077, Y  +709.719, Z    +0.000, E1   -21.590, E3 +284754.657}
SPL {X  -164.499, Y  +694.994, Z    +0.000, E1   -13.860, E3 +284755.442}
SPL {X  -165.382, Y  +684.927, Z    +0.000, E1    -7.984, E3 +284753.619}
SPL {X  -165.645, Y  +676.778, Z    +0.000, E1    -2.777, E3 +284753.341}
SPL {X  -165.650, Y  +672.041, Z    +0.000, E1    +0.844, E3 +284752.033}
SPL {X  -165.650, Y  +667.328, Z    +0.000, E1    +5.806, E3 +284751.410}
SPL {X  -165.650, Y  +661.774, Z    +0.000, E1   +13.006, E3 +284749.734}
SPL {X  -165.650, Y  +656.573, Z    +0.000, E1   +19.875, E3 +284750.292}
SPL {X  -165.650, Y  +650.769, Z    +0.000, E1   +28.083, E3 +284748.658}
SPL {X  -165.650, Y  +639.700, Z    +0.000, E1   +43.326, E3 +284743.720}
SPL {X  -165.650, Y  +605.320, Z    +0.000, E1   +76.562, E3 +284723.130}
SPL {X  -165.650, Y  +597.745, Z    +0.000, E1   +59.636, E3 +284761.131}
SPL {X  -165.650, Y  +596.360, Z    +0.000, E1   +54.978, E3 +284774.739}
SPL {X  -165.650, Y  +521.429, Z    +0.000, E1   +61.144, E3 +284827.970}
ENDSPLINE

SPLINE
SPL {X  -165.650, Y  +526.028, Z    +0.000, E1   +58.071, E3 +284841.745}
SPL {X  -165.650, Y  +539.856, Z    +0.000, E1   +53.398, E3 +284852.292}
ENDSPLINE

